METHOD PRIVATE popup : BOOL
VAR_INPUT
END_VAR
CASE popupStep OF
0:
	IF length>0 AND bSendCondition THEN
		_PopupLength:=length;
		popupSendData:=sendDataArray[cNumBegin];
		FOR iPopup:=cNumBegin TO (_PopupLength-1) DO
			sendDataArray[iPopup]:=sendDataArray[iPopup+1];
		END_FOR
		endPoint:=endPoint-1;
		length:=endPoint-cNumBegin;
		sendData(popupSendData);//此处是调用信息发送
		popupStep:=10;
	END_IF
10:
	popupTON2(IN:=NOT popupTON2.Q, PT:=T#2S);
	IF NOT bSendCondition OR popupTON2.Q THEN
		popupTON2(IN:=FALSE);
		popupStep:=11;
	END_IF
11:
	IF bSendCondition THEN
		popupStep:=12;
	END_IF
	popupTON1(IN:=FALSE);
12:
	//popupTON1(IN:=NOT popupTON1.Q,PT:=T#10MS);
	popupTON1(IN:=NOT popupTON1.Q,PT:=TO_TIME(nQueueInterval));
	IF popupTON1.Q THEN
		popupStep:=0;
	END_IF
END_CASE
END_METHOD

METHOD PRIVATE sendData : BOOL
VAR_INPUT
	dataStruct	:STRING(255);
END_VAR
IF bSendCondition AND bEnable THEN
	tcpipSendData:=dataStruct;
	
	CASE nSocketType OF
	0://TCPIP server
		tcpipSendDataBuff_Server:=tcpipSendData;
		tcpipSendData:=tcpipSendDataClear;	
		tcpipServer.bSend:=TRUE;
	1://TCPIP client
		tcpipSendDataBuff_Client:=tcpipSendData;
		tcpipSendData:=tcpipSendDataClear;	
		tcpipClient.bSend:=TRUE;
	END_CASE
	
	FOR logHandleArray_index:=1 TO logHandleArrayLength DO
		CASE nSocketType OF
		0://TCPIP server
			logHandleArray[logHandleArray_index]^.append(CONCAT(CONCAT(CONCAT('Send To ', sTerminalName), ' -- '),tcpipSendDataBuff_Server));
		1://TCPIP client
			logHandleArray[logHandleArray_index]^.append(CONCAT(CONCAT(CONCAT('Send To ', sTerminalName), ' -- '),tcpipSendDataBuff_Client));
		END_CASE
	END_FOR
END_IF
END_METHOD

END_PROGRAM

// ---- POUs/BaseModule/EL2252_2262Control/FlipperModule_EL2252.TcPOU
FUNCTION_BLOCK FlipperModule_EL2252
VAR CONSTANT
	gMaxPosNum								:INT:=100;
END_VAR
VAR_IN_OUT
	RefAxis_Ch1								:AXIS_REF;//ch1 运动主轴
	RemAxis_Ch1								:AXIS_REF;//ch1 锁存主轴
	RefAxis_Ch2								:AXIS_REF;//ch2 运动主轴
	RemAxis_Ch2								:AXIS_REF;//ch2 锁存主轴
END_VAR
VAR_INPUT
	FlipperOut1Times						:INT;//ch1 位置检测次数
	EnableOut1								:BOOL;//ch1 启用检测
	Out1_CamSwitchData						:ARRAY [1..gMaxPosNum] OF ST_CamSwitch;
	ForceOut1								:BOOL:=FALSE;//ch1 强制触发

	FlipperOut2Times						:INT;//ch2 位置检测次数
	EnableOut2								:BOOL;//ch2 启用检测
	ForceOut2								:BOOL:=FALSE;//ch2 强制触发
	Out2_CamSwitchData						:ARRAY [1..gMaxPosNum] OF ST_CamSwitch;
END_VAR
VAR_OUTPUT
	Out1RecPosArray1						:ARRAY [1..gMaxPosNum] OF LREAL:=[gMaxPosNum(0)];
	Out2RecPosArray2						:ARRAY [1..gMaxPosNum] OF LREAL:=[gMaxPosNum(0)];
	Ch1_LogOut								:STRING(255);
	Ch2_LogOut								:STRING(255);
	Io_EL2252								:EL2252_IoInterface;//硬件IO，需要关联至EL2252
	Ch1_Io_EL1252							:EL1252_IoInterface;//硬件IO，需要关联至EL1252
	Ch2_Io_EL1252							:EL1252_IoInterface;//硬件IO，需要关联至EL1252
END_VAR
VAR
//********************  XFC Calculate  *************************************************//
	Ch1_MC_DigitalCamSwitch					:MC_DigitalCamSwitch;
	Ch1_CAMSWITCH_REF						:CAMSWITCH_REF;
	Ch1_ArrMC_CamSwitch						:ARRAY [1..gMaxPosNum] OF MC_CamSwitch;
	Ch1_OUTPUT_REF							:OUTPUT_REF;
	Ch1_ST_CamSwitchOptions					:ST_CamSwitchOptions;
	Ch1_TRACK_REF							:TRACK_REF;

	Ch1_v									:INT:=0;//for CamswitchArray instance FirstPos and LastPos

	Ch2_MC_DigitalCamSwitch					:MC_DigitalCamSwitch;
	Ch2_CAMSWITCH_REF						:CAMSWITCH_REF;
	Ch2_ArrMC_CamSwitch						:ARRAY [1..gMaxPosNum] OF MC_CamSwitch;
	Ch2_OUTPUT_REF							:OUTPUT_REF;
	Ch2_ST_CamSwitchOptions					:ST_CamSwitchOptions;
	Ch2_TRACK_REF							:TRACK_REF;
	
	Ch2_v									:INT:=0;//for CamswitchArray instance FirstPos and LastPos
//********************  EL2252  *************************************************//
	Flipper_XFC_EL2252_V2					:XFC_EL2252_V2;
//****************************** XFC_touchprobe & EL1252  **********************//
	Ch1_XFC_TouchProbe						:XFC_TouchProbe;
	Ch1_ST_XfcTouchProbeOptions				:ST_XfcTouchProbeOptions;
	Ch1_XFC_TRIGGER_REF						:XFC_TRIGGER_REF;

	Ch1_fRecPos								:LREAL;
	Ch1_RecTrig								:R_TRIG;
	Ch1_nRecTimes							:INT:=1;
	Ch1_i									:INT:=1;

	Ch2_XFC_TouchProbe						:XFC_TouchProbe;
	Ch2_ST_XfcTouchProbeOptions				:ST_XfcTouchProbeOptions;
	Ch2_XFC_TRIGGER_REF						:XFC_TRIGGER_REF;

	Ch2_fRecPos								:LREAL;
	Ch2_RecTrig								:R_TRIG;
	Ch2_nRecTimes							:INT:=1;
	Ch2_i									:INT:=0;
	
	Ch1_LogFtrig							:F_TRIG;
	Ch1_LogRtrig							:R_TRIG;
	Ch1ClearI								:INT;
	Ch2_LogFtrig							:F_TRIG;
	Ch2_LogRtrig							:R_TRIG;
	Ch2ClearI								:INT;
END_VAR


//******************** Flipper Pos ****************************//
FOR Ch1_v:=1 TO FlipperOut1Times BY 1 DO
	Ch1_ArrMC_CamSwitch[Ch1_v].FirstOnPosition:=Out1_CamSwitchData[Ch1_v].fFirstOnPosition;
	Ch1_ArrMC_CamSwitch[Ch1_v].LastOnPosition:=Out1_CamSwitchData[Ch1_v].fLastOnPosition;//Out1PosS[Ch1_v]+1.5, Out1PosE[Ch1_v]
	
	IF Out1_CamSwitchData[Ch1_v].bTimeMode THEN
		Out1_CamSwitchData[Ch1_v].iAxisDirection:=0;
		Ch1_ArrMC_CamSwitch[Ch1_v].CamSwitchMode:=E_CamSwitchMode.CAMSWITCHMODE_TIME;//用时间模式可以通过 Duration 参数控制ON持续时间
		Ch1_ArrMC_CamSwitch[Ch1_v].Duration:=Out1_CamSwitchData[Ch1_v].fDuration;//持续时间, 单位s
	ELSE
		Ch1_ArrMC_CamSwitch[Ch1_v].CamSwitchMode:=E_CamSwitchMode.CAMSWITCHMODE_POSITION;//用位置模式可以通过 FirstOnPosition和LastOnPosition 参数控制ON持续时间
	END_IF
	IF 0>Out1_CamSwitchData[Ch1_v].iAxisDirection THEN
		Ch1_ArrMC_CamSwitch[Ch1_v].AxisDirection:=E_CamSwitchDirection.CAMSWITCHDIRECTION_NEGATIVE;
	ELSIF 0=Out1_CamSwitchData[Ch1_v].iAxisDirection THEN
		Ch1_ArrMC_CamSwitch[Ch1_v].AxisDirection:=E_CamSwitchDirection.CAMSWITCHDIRECTION_BOTH;
	ELSE
		Ch1_ArrMC_CamSwitch[Ch1_v].AxisDirection:=E_CamSwitchDirection.CAMSWITCHDIRECTION_POSITIVE;
	END_IF
END_FOR
Ch1_CAMSWITCH_REF.NumberOfSwitches:=TO_UDINT(FlipperOut1Times);
Ch1_CAMSWITCH_REF.pSwitches:=ADR(Ch1_ArrMC_CamSwitch);
Ch1_CAMSWITCH_REF.SizeOfSwitches:=SIZEOF(Ch1_ArrMC_CamSwitch);

FOR Ch2_v:=1 TO FlipperOut2Times BY 1 DO
	Ch2_ArrMC_CamSwitch[Ch2_v].FirstOnPosition:=Out2_CamSwitchData[Ch2_v].fFirstOnPosition;
	Ch2_ArrMC_CamSwitch[Ch2_v].LastOnPosition:=Out2_CamSwitchData[Ch2_v].fLastOnPosition;//Out2PosS[Ch2_v]+1.5, Out2PosE[Ch2_v]
	
	IF Out2_CamSwitchData[Ch2_v].bTimeMode THEN
		Out2_CamSwitchData[Ch2_v].iAxisDirection:=0;
		Ch2_ArrMC_CamSwitch[Ch2_v].CamSwitchMode:=E_CamSwitchMode.CAMSWITCHMODE_TIME;//用时间模式可以通过 Duration 参数控制ON持续时间
		Ch2_ArrMC_CamSwitch[Ch2_v].Duration:=Out2_CamSwitchData[Ch2_v].fDuration;//持续时间, 单位s
	ELSE
		Ch2_ArrMC_CamSwitch[Ch2_v].CamSwitchMode:=E_CamSwitchMode.CAMSWITCHMODE_POSITION;//用位置模式可以通过 FirstOnPosition和LastOnPosition 参数控制ON持续时间
	END_IF
	IF 0>Out2_CamSwitchData[Ch2_v].iAxisDirection THEN
		Ch2_ArrMC_CamSwitch[Ch2_v].AxisDirection:=E_CamSwitchDirection.CAMSWITCHDIRECTION_NEGATIVE;
	ELSIF 0=Out2_CamSwitchData[Ch2_v].iAxisDirection THEN
		Ch2_ArrMC_CamSwitch[Ch2_v].AxisDirection:=E_CamSwitchDirection.CAMSWITCHDIRECTION_BOTH;
	ELSE
		Ch2_ArrMC_CamSwitch[Ch2_v].AxisDirection:=E_CamSwitchDirection.CAMSWITCHDIRECTION_POSITIVE;
	END_IF
END_FOR
Ch2_CAMSWITCH_REF.NumberOfSwitches:=TO_UDINT(FlipperOut2Times);
Ch2_CAMSWITCH_REF.pSwitches:=ADR(Ch2_ArrMC_CamSwitch);
Ch2_CAMSWITCH_REF.SizeOfSwitches:=SIZEOF(Ch2_ArrMC_CamSwitch);
//******************** Cyclic IO ****************************//
EL1252();
EL2252V2();

METHOD PRIVATE EL1252
VAR_INPUT
END_VAR
//****************************** out1 EL1252 ***************************************//
Ch1_ST_XfcTouchProbeOptions.UseAcceleration:=TRUE;

Ch1_XFC_TRIGGER_REF.Signal:=Ch1_Io_EL1252.Input;
Ch1_XFC_TRIGGER_REF.TimestampRisingEdge:=Ch1_Io_EL1252.TimeStampNeg.dwLowPart;
Ch1_XFC_TRIGGER_REF.TimestampFallingEdge:=Ch1_Io_EL1252.TimeStampPos.dwLowPart;
Ch1_XFC_TRIGGER_REF.Edge:=E_SignalEdge.FallingEdge;
Ch1_XFC_TRIGGER_REF.FreeRun:=TRUE;
Ch1_XFC_TRIGGER_REF.ModuloPositions:=FALSE;
Ch1_XFC_TRIGGER_REF.EncoderIndex:=0;//DWORD_TO_UINT(RemAxis.NcToPlc.AxisId);

Ch1_XFC_TouchProbe(
	Axis:=RemAxis_Ch1 , 
	TriggerInput:=Ch1_XFC_TRIGGER_REF , 
	Execute:=TRUE , 
	WindowOnly:=FALSE , 
	FirstPosition:=0 , 
	LastPosition:=0 , 
	Options:=Ch1_ST_XfcTouchProbeOptions , 
	Done=> , 
	Busy=> , 
	Error=> , 
	ErrorID=> , 
	RecordedPosition=>Ch1_fRecPos );

Ch1_RecTrig(clk:=Ch1_XFC_TouchProbe.Done);
IF EnableOut1 THEN
	IF Ch1_RecTrig.Q THEN
		out1RecPosArray1[Ch1_nRecTimes]:=Ch1_fRecPos;
		Ch1_nRecTimes:=Ch1_nRecTimes+1;
	END_IF
END_IF

Ch1_LogRtrig(clk:=EnableOut1);
IF Ch1_LogRtrig.Q THEN
	FOR Ch1ClearI:=1 TO gMaxPosNum DO
		out1RecPosArray1[Ch1ClearI]:=0;
	END_FOR
END_IF

Ch1_LogFtrig(clk:=EnableOut1);
IF Ch1_LogFtrig.Q THEN
	Ch1_LogOut:='out1 Pos: ';
	FOR Ch1_i:=1 TO FlipperOut1Times BY 1 DO
		Ch1_LogOut:=concat(Ch1_LogOut,LREAL_TO_STRING(out1RecPosArray1[Ch1_i]));
		Ch1_LogOut:=concat(Ch1_LogOut,' ');
	END_FOR
	Ch1_nRecTimes:=1;
END_IF
//****************************** out2 EL1252 ***************************************//
Ch2_ST_XfcTouchProbeOptions.UseAcceleration:=TRUE;

Ch2_XFC_TRIGGER_REF.Signal:=Ch2_Io_EL1252.Input;
Ch2_XFC_TRIGGER_REF.TimestampRisingEdge:=Ch2_Io_EL1252.TimeStampNeg.dwLowPart;
Ch2_XFC_TRIGGER_REF.TimestampFallingEdge:=Ch2_Io_EL1252.TimeStampPos.dwLowPart;
Ch2_XFC_TRIGGER_REF.Edge:=E_SignalEdge.FallingEdge;
Ch2_XFC_TRIGGER_REF.FreeRun:=TRUE;
Ch2_XFC_TRIGGER_REF.ModuloPositions:=FALSE;
Ch2_XFC_TRIGGER_REF.EncoderIndex:=0;//DWORD_TO_UINT(RemAxis.NcToPlc.AxisId);

Ch2_XFC_TouchProbe(
	Axis:=RemAxis_Ch2 , 
	TriggerInput:=Ch2_XFC_TRIGGER_REF , 
	Execute:=TRUE , 
	WindowOnly:=FALSE , 
	FirstPosition:=0 , 
	LastPosition:=0 , 
	Options:=Ch2_ST_XfcTouchProbeOptions , 
	Done=> , 
	Busy=> , 
	Error=> , 
	ErrorID=> , 
	RecordedPosition=>Ch2_fRecPos );

Ch2_RecTrig(clk:=Ch2_XFC_TouchProbe.Done);
IF EnableOut2 THEN
	IF Ch2_RecTrig.Q THEN
		out2RecPosArray2[Ch2_nRecTimes]:=Ch2_fRecPos;
		Ch2_nRecTimes:=Ch2_nRecTimes+1;
	END_IF
END_IF

Ch2_LogRtrig(clk:=EnableOut2);
IF Ch2_LogRtrig.Q THEN
	FOR Ch2ClearI:=1 TO gMaxPosNum DO
		Out2RecPosArray2[Ch2ClearI]:=0;
	END_FOR
END_IF

Ch2_LogFtrig(clk:=EnableOut2);
IF Ch2_LogFtrig.Q THEN
	Ch2_LogOut:='out2 Pos: ';
	FOR Ch2_i:=1 TO FlipperOut2Times BY 1 DO
		Ch2_LogOut:=concat(Ch2_LogOut,LREAL_TO_STRING(out2RecPosArray2[Ch2_i]));
		Ch2_LogOut:=concat(Ch2_LogOut,' ');
	END_FOR
	Ch2_nRecTimes:=1;
END_IF
END_METHOD

METHOD PRIVATE EL2252V2
VAR_INPUT
END_VAR
//*******************   output 1  *****************************//
Ch1_ST_CamSwitchOptions.EncoderIndex:=0;//DWORD_TO_UINT(RefAxis.NcToPlc.AxisId);
Ch1_ST_CamSwitchOptions.UseAcceleration:=TRUE;

Ch1_TRACK_REF.ModuloPositions:=FALSE;//启用 模位置
Ch1_TRACK_REF.Disable:=FALSE;
Ch1_TRACK_REF.Force:=ForceOut1;
Ch1_TRACK_REF.OnCompensation:=0;//延时 ON
Ch1_TRACK_REF.OffCompensation:=0;//延时 OFF

Ch1_MC_DigitalCamSwitch(
	Axis:=RefAxis_Ch1 , 
	Switches:=Ch1_CAMSWITCH_REF , 
	Output:=Ch1_OUTPUT_REF , 
	TrackOptions:=Ch1_TRACK_REF , 
	Enable:=EnableOut1 , 
	Options:=Ch1_ST_CamSwitchOptions , 
	InOperation=> , 
	Busy=> , 
	Error=> , 
	ErrorID=> );

//*******************   output 2  *****************************//
Ch2_ST_CamSwitchOptions.EncoderIndex:=0;//DWORD_TO_UINT(RefAxis.NcToPlc.AxisId);
Ch2_ST_CamSwitchOptions.UseAcceleration:=TRUE;

Ch2_TRACK_REF.ModuloPositions:=FALSE;//启用 模位置
Ch2_TRACK_REF.Disable:=FALSE;
Ch2_TRACK_REF.Force:=ForceOut2;
Ch2_TRACK_REF.OnCompensation:=0;//延时 ON
Ch2_TRACK_REF.OffCompensation:=0;//延时 OFF

Ch2_MC_DigitalCamSwitch(
	Axis:=RefAxis_Ch2 , 
	Switches:=Ch2_CAMSWITCH_REF , 
	Output:=Ch2_OUTPUT_REF , 
	TrackOptions:=Ch2_TRACK_REF , 
	Enable:=EnableOut2 , 
	Options:=Ch2_ST_CamSwitchOptions , 
	InOperation=> , 
	Busy=> , 
	Error=> , 
	ErrorID=> );

//***************** EL2252 *****************************//
Flipper_XFC_EL2252_V2(
	ForceWhenLate:=TRUE , 
	Error=> , 
	ErrorID=> , 
	ErrorOutputMissed=> , 
	PrecisionReduced=> , 
	Output1:=Ch1_OUTPUT_REF , 
	Output2:=Ch2_OUTPUT_REF , 
	TrackOptions1:=Ch1_TRACK_REF , 
	TrackOptions2:=Ch2_TRACK_REF , 
	EL2252:=Io_EL2252 );
END_METHOD

METHOD SetCamSwitchData_Ch1 : BOOL
VAR_INPUT
	nIndex:INT;
	
	bTimeMode:BOOL;//TRUE表示时间控制模式, 持续时间由fDuration控制; FALSE表示位置控制模式，持续时间由fFirstOnPosition和fLastOnPosition控制
	fDuration:LREAL;//持续时间, 单位s
	
	fFirstOnPosition:LREAL;//时间控制模式和位置控制模式触发起始点
	fLastOnPosition:LREAL;//位置控制模式触发结束点
	iAxisDirection:INT;//-1表示负方向检测; 0表示正负方向检测(时间控制模式必须是0); 1表示正方向检测;
END_VAR
IF nIndex<1 OR nIndex>gMaxPosNum THEN
	SetCamSwitchData_Ch1:=FALSE;
	RETURN;
END_IF
Out1_CamSwitchData[nIndex].bTimeMode:=bTimeMode;
Out1_CamSwitchData[nIndex].fDuration:=fDuration;
Out1_CamSwitchData[nIndex].fFirstOnPosition:=fFirstOnPosition;
Out1_CamSwitchData[nIndex].fLastOnPosition:=fLastOnPosition;
Out1_CamSwitchData[nIndex].iAxisDirection:=iAxisDirection;
SetCamSwitchData_Ch1:=TRUE;
END_METHOD

METHOD SetCamSwitchData_Ch2 : BOOL
VAR_INPUT
	nIndex:INT;
	
	bTimeMode:BOOL;//TRUE表示时间控制模式, 持续时间由fDuration控制; FALSE表示位置控制模式，持续时间由fFirstOnPosition和fLastOnPosition控制
	fDuration:LREAL;//持续时间, 单位s
	
	fFirstOnPosition:LREAL;//时间控制模式和位置控制模式触发起始点
	fLastOnPosition:LREAL;//位置控制模式触发结束点
	iAxisDirection:INT;//-1表示负方向检测; 0表示正负方向检测(时间控制模式必须是0); 1表示正方向检测;
END_VAR
IF nIndex<1 OR nIndex>gMaxPosNum THEN
	SetCamSwitchData_Ch2:=FALSE;
	RETURN;
END_IF
Out2_CamSwitchData[nIndex].bTimeMode:=bTimeMode;
Out2_CamSwitchData[nIndex].fDuration:=fDuration;
Out2_CamSwitchData[nIndex].fFirstOnPosition:=fFirstOnPosition;
Out2_CamSwitchData[nIndex].fLastOnPosition:=fLastOnPosition;
Out2_CamSwitchData[nIndex].iAxisDirection:=iAxisDirection;
SetCamSwitchData_Ch2:=TRUE;
END_METHOD

ACTION VersionLog:
(*
版本: V1.0.0.0
说明:
	1. 首个版本
/**************************************************/
版本: V1.0.0.1
说明:
	1. 增加触发上升沿清空EL1252位置记录数据
/**************************************************/
版本: V1.0.0.2
说明:
	1. 增加函数接口，用于设置飞拍监控数据
/**************************************************/
*)
END_ACTION

END_FUNCTION_BLOCK

// ---- POUs/BaseModule/EL2252_2262Control/FlipperModule_EL2262.TcPOU
FUNCTION_BLOCK FlipperModule_EL2262
VAR CONSTANT
	gMaxPosNum								:INT:=100;
END_VAR
VAR_IN_OUT
	RefAxis_Ch1								:AXIS_REF;//ch1 运动主轴
	RemAxis_Ch1								:AXIS_REF;//ch1 锁存主轴
	RefAxis_Ch2								:AXIS_REF;//ch2 运动主轴
	RemAxis_Ch2								:AXIS_REF;//ch2 锁存主轴
END_VAR
VAR_INPUT
	OversamplingFactor						:UINT:=1000;// 超采样因子, Operation Mode需要设置成2 Channels(Bytes)
	FlipperOut1Times						:INT;//ch1 位置检测次数
	EnableOut1								:BOOL;//ch1 启用检测
	Out1_CamSwitchData						:ARRAY [1..gMaxPosNum] OF ST_CamSwitch_EL2262;
	ForceOut1								:BOOL:=FALSE;//ch1 强制触发

	FlipperOut2Times						:INT;//ch2 位置检测次数
	EnableOut2								:BOOL;//ch2 启用检测
	Out2_CamSwitchData						:ARRAY [1..gMaxPosNum] OF ST_CamSwitch_EL2262;
	ForceOut2								:BOOL:=FALSE;//ch2 强制触发
END_VAR
VAR_OUTPUT
	Out1RecPosArray1						:ARRAY [1..gMaxPosNum] OF LREAL:=[gMaxPosNum(0)];//记录锁存触发位置数组
	Out2RecPosArray2						:ARRAY [1..gMaxPosNum] OF LREAL:=[gMaxPosNum(0)];//记录锁存触发位置数组
	Ch1_LogOut								:STRING(255);
	Ch2_LogOut								:STRING(255);
	Io_EL2262								:EL2262_IoInterface;//硬件IO，需要关联至EL2262
	Io_EL2262_Ch2							:EL2262_IoInterface;//硬件IO，需要关联至EL2262
	Ch1_Io_EL1252							:EL1252_IoInterface;//硬件IO，需要关联至EL1252
	Ch2_Io_EL1252							:EL1252_IoInterface;//硬件IO，需要关联至EL1252
END_VAR
VAR
//********************  XFC Calculate  *************************************************//
	Ch1_MC_DigitalCamSwitch					:MC_DigitalCamSwitch;
	Ch1_CAMSWITCH_REF						:CAMSWITCH_REF;
	Ch1_ArrMC_CamSwitch						:ARRAY [1..gMaxPosNum] OF MC_CamSwitch;
	Ch1_OUTPUT_REF							:OUTPUT_REF;
	Ch1_ST_CamSwitchOptions					:ST_CamSwitchOptions;
	Ch1_TRACK_REF							:TRACK_REF;

	Ch1_v									:INT:=0;//for CamswitchArray instance FirstPos and LastPos

	Ch2_MC_DigitalCamSwitch					:MC_DigitalCamSwitch;
	Ch2_CAMSWITCH_REF						:CAMSWITCH_REF;
	Ch2_ArrMC_CamSwitch						:ARRAY [1..gMaxPosNum] OF MC_CamSwitch;
	Ch2_OUTPUT_REF							:OUTPUT_REF;
	Ch2_ST_CamSwitchOptions					:ST_CamSwitchOptions;
	Ch2_TRACK_REF							:TRACK_REF;
	
	Ch2_v									:INT:=0;//for CamswitchArray instance FirstPos and LastPos
//********************  EL2252  *************************************************//
	Flipper_CH1_XFC_EL2262					:XFC_EL2262;
	Flipper_CH2_XFC_EL2262					:XFC_EL2262;
	
//****************************** XFC_touchprobe & EL1252  **********************//
	Ch1_XFC_TouchProbe						:XFC_TouchProbe;
	Ch1_ST_XfcTouchProbeOptions				:ST_XfcTouchProbeOptions;
	Ch1_XFC_TRIGGER_REF						:XFC_TRIGGER_REF;

	Ch1_fRecPos								:LREAL;
	Ch1_RecTrig								:R_TRIG;
	Ch1_nRecTimes							:INT:=1;//用于记录锁存触发次数
	Ch1_i									:INT:=1;

	Ch2_XFC_TouchProbe						:XFC_TouchProbe;
	Ch2_ST_XfcTouchProbeOptions				:ST_XfcTouchProbeOptions;
	Ch2_XFC_TRIGGER_REF						:XFC_TRIGGER_REF;

	Ch2_fRecPos								:LREAL;
	Ch2_RecTrig								:R_TRIG;
	Ch2_nRecTimes							:INT:=1;//用于记录锁存触发次数
	Ch2_i									:INT:=0;
	
	Ch1_LogFtrig							:F_TRIG;
	Ch1_LogRtrig							:R_TRIG;
	Ch1ClearI								:INT;
	Ch2_LogFtrig							:F_TRIG;
	Ch2_LogRtrig							:R_TRIG;
	Ch2ClearI								:INT;
END_VAR


//******************** Flipper Pos ****************************//
FOR Ch1_v:=1 TO FlipperOut1Times BY 1 DO
	Ch1_ArrMC_CamSwitch[Ch1_v].FirstOnPosition:=Out1_CamSwitchData[Ch1_v].fFirstOnPosition;
	Ch1_ArrMC_CamSwitch[Ch1_v].LastOnPosition:=Out1_CamSwitchData[Ch1_v].fLastOnPosition;//Out1PosS[Ch1_v]+1.5, Out1PosE[Ch1_v]
	
	IF Out1_CamSwitchData[Ch1_v].bTimeMode THEN
		Out1_CamSwitchData[Ch1_v].iAxisDirection:=0;
		Ch1_ArrMC_CamSwitch[Ch1_v].CamSwitchMode:=E_CamSwitchMode.CAMSWITCHMODE_TIME;//用时间模式可以通过 Duration 参数控制ON持续时间
		Ch1_ArrMC_CamSwitch[Ch1_v].Duration:=Out1_CamSwitchData[Ch1_v].fDuration;//持续时间, 单位s
	ELSE
		Ch1_ArrMC_CamSwitch[Ch1_v].CamSwitchMode:=E_CamSwitchMode.CAMSWITCHMODE_POSITION;//用位置模式可以通过 FirstOnPosition和LastOnPosition 参数控制ON持续时间
	END_IF
	IF 0>Out1_CamSwitchData[Ch1_v].iAxisDirection THEN
		Ch1_ArrMC_CamSwitch[Ch1_v].AxisDirection:=E_CamSwitchDirection.CAMSWITCHDIRECTION_NEGATIVE;
	ELSIF 0=Out1_CamSwitchData[Ch1_v].iAxisDirection THEN
		Ch1_ArrMC_CamSwitch[Ch1_v].AxisDirection:=E_CamSwitchDirection.CAMSWITCHDIRECTION_BOTH;
	ELSE
		Ch1_ArrMC_CamSwitch[Ch1_v].AxisDirection:=E_CamSwitchDirection.CAMSWITCHDIRECTION_POSITIVE;
	END_IF
	
	(*Ch1_ArrMC_CamSwitch[Ch1_v].CamSwitchMode:=E_CamSwitchMode.CAMSWITCHMODE_POSITION;//用位置模式可以通过 FirstOnPosition和LastOnPosition 参数控制ON持续时间
	IF 0>Out1_CamSwitchData[Ch1_v].iAxisDirection THEN
		Ch1_ArrMC_CamSwitch[Ch1_v].AxisDirection:=E_CamSwitchDirection.CAMSWITCHDIRECTION_NEGATIVE;
	ELSIF 0=Out1_CamSwitchData[Ch1_v].iAxisDirection THEN
		Ch1_ArrMC_CamSwitch[Ch1_v].AxisDirection:=E_CamSwitchDirection.CAMSWITCHDIRECTION_BOTH;
	ELSE
		Ch1_ArrMC_CamSwitch[Ch1_v].AxisDirection:=E_CamSwitchDirection.CAMSWITCHDIRECTION_POSITIVE;
	END_IF*)
END_FOR
Ch1_CAMSWITCH_REF.NumberOfSwitches:=TO_UDINT(FlipperOut1Times);
Ch1_CAMSWITCH_REF.pSwitches:=ADR(Ch1_ArrMC_CamSwitch);
Ch1_CAMSWITCH_REF.SizeOfSwitches:=SIZEOF(Ch1_ArrMC_CamSwitch);

FOR Ch2_v:=1 TO FlipperOut2Times BY 1 DO
	Ch2_ArrMC_CamSwitch[Ch2_v].FirstOnPosition:=Out2_CamSwitchData[Ch2_v].fFirstOnPosition;
	Ch2_ArrMC_CamSwitch[Ch2_v].LastOnPosition:=Out2_CamSwitchData[Ch2_v].fLastOnPosition;//Out2PosS[Ch2_v]+1.5, Out2PosE[Ch2_v]
	
	IF Out2_CamSwitchData[Ch2_v].bTimeMode THEN
		Out2_CamSwitchData[Ch2_v].iAxisDirection:=0;
		Ch2_ArrMC_CamSwitch[Ch2_v].CamSwitchMode:=E_CamSwitchMode.CAMSWITCHMODE_TIME;//用时间模式可以通过 Duration 参数控制ON持续时间
		Ch2_ArrMC_CamSwitch[Ch2_v].Duration:=Out2_CamSwitchData[Ch2_v].fDuration;//持续时间, 单位s
	ELSE
		Ch2_ArrMC_CamSwitch[Ch2_v].CamSwitchMode:=E_CamSwitchMode.CAMSWITCHMODE_POSITION;//用位置模式可以通过 FirstOnPosition和LastOnPosition 参数控制ON持续时间
	END_IF
	IF 0>Out2_CamSwitchData[Ch2_v].iAxisDirection THEN
		Ch2_ArrMC_CamSwitch[Ch2_v].AxisDirection:=E_CamSwitchDirection.CAMSWITCHDIRECTION_NEGATIVE;
	ELSIF 0=Out2_CamSwitchData[Ch2_v].iAxisDirection THEN
		Ch2_ArrMC_CamSwitch[Ch2_v].AxisDirection:=E_CamSwitchDirection.CAMSWITCHDIRECTION_BOTH;
	ELSE
		Ch2_ArrMC_CamSwitch[Ch2_v].AxisDirection:=E_CamSwitchDirection.CAMSWITCHDIRECTION_POSITIVE;
	END_IF
	
	(*Ch2_ArrMC_CamSwitch[Ch2_v].CamSwitchMode:=E_CamSwitchMode.CAMSWITCHMODE_POSITION;//用位置模式可以通过 FirstOnPosition和LastOnPosition 参数控制ON持续时间
	IF 0>Out2_CamSwitchData[Ch2_v].iAxisDirection THEN
		Ch2_ArrMC_CamSwitch[Ch2_v].AxisDirection:=E_CamSwitchDirection.CAMSWITCHDIRECTION_NEGATIVE;
	ELSIF 0=Out2_CamSwitchData[Ch2_v].iAxisDirection THEN
		Ch2_ArrMC_CamSwitch[Ch2_v].AxisDirection:=E_CamSwitchDirection.CAMSWITCHDIRECTION_BOTH;
	ELSE
		Ch2_ArrMC_CamSwitch[Ch2_v].AxisDirection:=E_CamSwitchDirection.CAMSWITCHDIRECTION_POSITIVE;
	END_IF*)
END_FOR
Ch2_CAMSWITCH_REF.NumberOfSwitches:=TO_UDINT(FlipperOut2Times);
Ch2_CAMSWITCH_REF.pSwitches:=ADR(Ch2_ArrMC_CamSwitch);
Ch2_CAMSWITCH_REF.SizeOfSwitches:=SIZEOF(Ch2_ArrMC_CamSwitch);
//******************** Cyclic IO ****************************//
EL2262();
EL1252();

METHOD PRIVATE EL1252
VAR_INPUT
END_VAR
//****************************** out1 EL1252 ***************************************//
Ch1_ST_XfcTouchProbeOptions.UseAcceleration:=TRUE;
(*
Ch1_XFC_TRIGGER_REF.Signal:=Ch1_Io_EL1252.Input;
Ch1_XFC_TRIGGER_REF.TimestampRisingEdge:=Ch1_Io_EL1252.TimeStampNeg.dwLowPart;
Ch1_XFC_TRIGGER_REF.TimestampFallingEdge:=Ch1_Io_EL1252.TimeStampPos.dwLowPart;
Ch1_XFC_TRIGGER_REF.Edge:=E_SignalEdge.FallingEdge;
Ch1_XFC_TRIGGER_REF.FreeRun:=TRUE;
Ch1_XFC_TRIGGER_REF.ModuloPositions:=FALSE;
Ch1_XFC_TRIGGER_REF.EncoderIndex:=0;//DWORD_TO_UINT(RemAxis.NcToPlc.AxisId);
*)
Ch1_XFC_TRIGGER_REF.Signal:=Ch1_Io_EL1252.Input;
Ch1_XFC_TRIGGER_REF.TimestampRisingEdge:=Ch1_Io_EL1252.TimeStampPos.dwLowPart;
Ch1_XFC_TRIGGER_REF.TimestampFallingEdge:=Ch1_Io_EL1252.TimeStampNeg.dwLowPart;
Ch1_XFC_TRIGGER_REF.Edge:=E_SignalEdge.RisingEdge;
Ch1_XFC_TRIGGER_REF.FreeRun:=TRUE;
Ch1_XFC_TRIGGER_REF.ModuloPositions:=FALSE;
Ch1_XFC_TRIGGER_REF.EncoderIndex:=0;//DWORD_TO_UINT(RemAxis_Ch1.NcToPlc.AxisId);

RemAxis_Ch1.ReadStatus();
Ch1_XFC_TouchProbe(
	Axis:=RemAxis_Ch1 , 
	TriggerInput:=Ch1_XFC_TRIGGER_REF , 
	Execute:=TRUE , 
	WindowOnly:=FALSE , 
	FirstPosition:=0 , 
	LastPosition:=0 , 
	Options:=Ch1_ST_XfcTouchProbeOptions , 
	Done=> , 
	Busy=> , 
	Error=> , 
	ErrorID=> , 
	RecordedPosition=>Ch1_fRecPos );

Ch1_RecTrig(clk:=Ch1_XFC_TouchProbe.Done);
IF EnableOut1 THEN
	IF Ch1_RecTrig.Q THEN
		out1RecPosArray1[Ch1_nRecTimes]:=Ch1_fRecPos;
		Ch1_nRecTimes:=Ch1_nRecTimes+1;
	END_IF
END_IF

Ch1_LogRtrig(clk:=EnableOut1);
IF Ch1_LogRtrig.Q THEN
	FOR Ch1ClearI:=1 TO gMaxPosNum DO
		out1RecPosArray1[Ch1ClearI]:=0;
	END_FOR
END_IF

Ch1_LogFtrig(clk:=EnableOut1);
IF Ch1_LogFtrig.Q THEN
	Ch1_LogOut:='out1 Pos:,';
	//FOR Ch1_i:=1 TO FlipperOut1Times BY 1 DO
	FOR Ch1_i:=1 TO (Ch1_nRecTimes-1) BY 1 DO
		//Ch1_LogOut:=concat(Ch1_LogOut,LREAL_TO_STRING(out1RecPosArray1[Ch1_i]));
		Ch1_LogOut:=concat(Ch1_LogOut,LREAL_TO_FMTSTR(out1RecPosArray1[Ch1_i],5,FALSE));
		Ch1_LogOut:=concat(Ch1_LogOut,',');
	END_FOR
	Ch1_nRecTimes:=1;
END_IF
//****************************** out2 EL1252 ***************************************//
Ch2_ST_XfcTouchProbeOptions.UseAcceleration:=TRUE;
(*
Ch2_XFC_TRIGGER_REF.Signal:=Ch2_Io_EL1252.Input;
Ch2_XFC_TRIGGER_REF.TimestampRisingEdge:=Ch2_Io_EL1252.TimeStampNeg.dwLowPart;
Ch2_XFC_TRIGGER_REF.TimestampFallingEdge:=Ch2_Io_EL1252.TimeStampPos.dwLowPart;
Ch2_XFC_TRIGGER_REF.Edge:=E_SignalEdge.FallingEdge;
Ch2_XFC_TRIGGER_REF.FreeRun:=TRUE;
Ch2_XFC_TRIGGER_REF.ModuloPositions:=FALSE;
Ch2_XFC_TRIGGER_REF.EncoderIndex:=0;//DWORD_TO_UINT(RemAxis.NcToPlc.AxisId);
*)
Ch2_XFC_TRIGGER_REF.Signal:=Ch2_Io_EL1252.Input;
Ch2_XFC_TRIGGER_REF.TimestampRisingEdge:=Ch2_Io_EL1252.TimeStampPos.dwLowPart;
Ch2_XFC_TRIGGER_REF.TimestampFallingEdge:=Ch2_Io_EL1252.TimeStampNeg.dwLowPart;
Ch2_XFC_TRIGGER_REF.Edge:=E_SignalEdge.RisingEdge;
Ch2_XFC_TRIGGER_REF.FreeRun:=TRUE;
Ch2_XFC_TRIGGER_REF.ModuloPositions:=FALSE;
Ch2_XFC_TRIGGER_REF.EncoderIndex:=0;//DWORD_TO_UINT(RemAxis_Ch2.NcToPlc.AxisId);

RemAxis_Ch2.ReadStatus();
Ch2_XFC_TouchProbe(
	Axis:=RemAxis_Ch2 , 
	TriggerInput:=Ch2_XFC_TRIGGER_REF , 
	Execute:=TRUE , 
	WindowOnly:=FALSE , 
	FirstPosition:=0 , 
	LastPosition:=0 , 
	Options:=Ch2_ST_XfcTouchProbeOptions , 
	Done=> , 
	Busy=> , 
	Error=> , 
	ErrorID=> , 
	RecordedPosition=>Ch2_fRecPos );


Ch2_RecTrig(clk:=Ch2_XFC_TouchProbe.Done);
IF EnableOut2 THEN
	IF Ch2_RecTrig.Q THEN
		out2RecPosArray2[Ch2_nRecTimes]:=Ch2_fRecPos;
		Ch2_nRecTimes:=Ch2_nRecTimes+1;
	END_IF
END_IF

Ch2_LogRtrig(clk:=EnableOut2);
IF Ch2_LogRtrig.Q THEN
	FOR Ch2ClearI:=1 TO gMaxPosNum DO
		Out2RecPosArray2[Ch2ClearI]:=0;
	END_FOR
END_IF

Ch2_LogFtrig(clk:=EnableOut2);
IF Ch2_LogFtrig.Q THEN
	Ch2_LogOut:='out2 Pos:,';
	//FOR Ch2_i:=1 TO FlipperOut2Times BY 1 DO
	FOR Ch2_i:=1 TO (Ch2_nRecTimes-1) BY 1 DO
		//Ch2_LogOut:=concat(Ch2_LogOut,LREAL_TO_STRING(out2RecPosArray2[Ch2_i]));
		Ch2_LogOut:=concat(Ch2_LogOut,LREAL_TO_FMTSTR(out2RecPosArray2[Ch2_i],5,FALSE));
		Ch2_LogOut:=concat(Ch2_LogOut,',');
	END_FOR
	Ch2_nRecTimes:=1;
END_IF
END_METHOD

METHOD PRIVATE EL2262
VAR_INPUT
END_VAR
//*******************   output 1  *****************************//
Ch1_ST_CamSwitchOptions.EncoderIndex:=0;//DWORD_TO_UINT(RefAxis.NcToPlc.AxisId);
Ch1_ST_CamSwitchOptions.UseAcceleration:=TRUE;//FALSE TRUE

Ch1_TRACK_REF.ModuloPositions:=FALSE;//启用 模位置
Ch1_TRACK_REF.Disable:=FALSE;
Ch1_TRACK_REF.Force:=ForceOut1;
Ch1_TRACK_REF.OnCompensation:=0;//延时 ON
Ch1_TRACK_REF.OffCompensation:=0;//延时 OFF

RefAxis_Ch1.ReadStatus();
Ch1_MC_DigitalCamSwitch(
	Axis:=RefAxis_Ch1 , 
	Switches:=Ch1_CAMSWITCH_REF , 
	Output:=Ch1_OUTPUT_REF , 
	TrackOptions:=Ch1_TRACK_REF , 
	Enable:=EnableOut1 , 
	Options:=Ch1_ST_CamSwitchOptions , 
	InOperation=> , 
	Busy=> , 
	Error=> , 
	ErrorID=> );
(*
IF RefAxis_Ch1.Status.NotMoving THEN
	Ch1_MC_DigitalCamSwitch(
		Axis:=RefAxis_Ch1 , 
		Switches:=Ch1_CAMSWITCH_REF , 
		Output:=Ch1_OUTPUT_REF , 
		TrackOptions:=Ch1_TRACK_REF , 
		Enable:=FALSE , 
		Options:=Ch1_ST_CamSwitchOptions , 
		InOperation=> , 
		Busy=> , 
		Error=> , 
		ErrorID=> );
END_IF
*)
//*******************   output 2  *****************************//
Ch2_ST_CamSwitchOptions.EncoderIndex:=0;//DWORD_TO_UINT(RefAxis.NcToPlc.AxisId);
Ch2_ST_CamSwitchOptions.UseAcceleration:=TRUE;//FALSE TRUE

Ch2_TRACK_REF.ModuloPositions:=FALSE;//启用 模位置
Ch2_TRACK_REF.Disable:=FALSE;
Ch2_TRACK_REF.Force:=ForceOut2;
Ch2_TRACK_REF.OnCompensation:=0;//延时 ON
Ch2_TRACK_REF.OffCompensation:=0;//延时 OFF

RefAxis_Ch2.ReadStatus();
Ch2_MC_DigitalCamSwitch(
	Axis:=RefAxis_Ch2 , 
	Switches:=Ch2_CAMSWITCH_REF , 
	Output:=Ch2_OUTPUT_REF , 
	TrackOptions:=Ch2_TRACK_REF , 
	Enable:=EnableOut2 , 
	Options:=Ch2_ST_CamSwitchOptions , 
	InOperation=> , 
	Busy=> , 
	Error=> , 
	ErrorID=> );
(*
IF RefAxis_Ch2.Status.NotMoving THEN
	Ch2_MC_DigitalCamSwitch(
		Axis:=RefAxis_Ch2 , 
		Switches:=Ch2_CAMSWITCH_REF , 
		Output:=Ch2_OUTPUT_REF , 
		TrackOptions:=Ch2_TRACK_REF , 
		Enable:=FALSE , 
		Options:=Ch2_ST_CamSwitchOptions , 
		InOperation=> , 
		Busy=> , 
		Error=> , 
		ErrorID=> );
END_IF
*)
//***************** EL2262 *****************************//
Flipper_CH1_XFC_EL2262(
	OversamplingFactor:= OversamplingFactor, 
	OutputOneCycleDelayed:= FALSE, 
	ForceWhenLate:= TRUE, 
	Channel:= 0, 
	Error=> , 
	ErrorID=> , 
	ErrorOutputMissed=> , 
	PrecisionReduced=> , 
	Output:= Ch1_OUTPUT_REF, 
	TrackOptions:= Ch1_TRACK_REF, 
	EL2262:= Io_EL2262);

Flipper_CH2_XFC_EL2262(
	OversamplingFactor:= OversamplingFactor, 
	OutputOneCycleDelayed:= FALSE, 
	ForceWhenLate:= TRUE, 
	Channel:= 1, 
	Error=> , 
	ErrorID=> , 
	ErrorOutputMissed=> , 
	PrecisionReduced=> , 
	Output:= Ch2_OUTPUT_REF, 
	TrackOptions:= Ch2_TRACK_REF, 
	EL2262:= Io_EL2262_Ch2);
END_METHOD

METHOD SetCamSwitchData_Ch1 : BOOL
VAR_INPUT
	nIndex:INT;
	
	bTimeMode:BOOL;//TRUE表示时间控制模式, 持续时间由fDuration控制; FALSE表示位置控制模式，持续时间由fFirstOnPosition和fLastOnPosition控制
	fDuration:LREAL;//持续时间, 单位s
	
	fFirstOnPosition:LREAL;//时间控制模式和位置控制模式触发起始点
	fLastOnPosition:LREAL;//位置控制模式触发结束点
	iAxisDirection:INT;//-1表示负方向检测; 0表示正负方向检测(时间控制模式必须是0); 1表示正方向检测;
END_VAR
IF nIndex<1 OR nIndex>gMaxPosNum THEN
	SetCamSwitchData_Ch1:=FALSE;
	RETURN;
END_IF
Out1_CamSwitchData[nIndex].bTimeMode:=bTimeMode;
Out1_CamSwitchData[nIndex].fDuration:=fDuration;
Out1_CamSwitchData[nIndex].fFirstOnPosition:=fFirstOnPosition;
Out1_CamSwitchData[nIndex].fLastOnPosition:=fLastOnPosition;
Out1_CamSwitchData[nIndex].iAxisDirection:=iAxisDirection;
SetCamSwitchData_Ch1:=TRUE;
END_METHOD

METHOD SetCamSwitchData_Ch2 : BOOL
VAR_INPUT
	nIndex:INT;
	
	bTimeMode:BOOL;//TRUE表示时间控制模式, 持续时间由fDuration控制; FALSE表示位置控制模式，持续时间由fFirstOnPosition和fLastOnPosition控制
	fDuration:LREAL;//持续时间, 单位s
	
	fFirstOnPosition:LREAL;//时间控制模式和位置控制模式触发起始点
	fLastOnPosition:LREAL;//位置控制模式触发结束点
	iAxisDirection:INT;//-1表示负方向检测; 0表示正负方向检测(时间控制模式必须是0); 1表示正方向检测;
END_VAR
IF nIndex<1 OR nIndex>gMaxPosNum THEN
	SetCamSwitchData_Ch2:=FALSE;
	RETURN;
END_IF
Out2_CamSwitchData[nIndex].bTimeMode:=bTimeMode;
Out2_CamSwitchData[nIndex].fDuration:=fDuration;
Out2_CamSwitchData[nIndex].fFirstOnPosition:=fFirstOnPosition;
Out2_CamSwitchData[nIndex].fLastOnPosition:=fLastOnPosition;
Out2_CamSwitchData[nIndex].iAxisDirection:=iAxisDirection;
SetCamSwitchData_Ch2:=TRUE;
END_METHOD

ACTION VersionLog:
(*
版本: V1.0.0.0
说明:
	1. 首个版本
/**************************************************/
版本: V1.0.0.1
说明:
	1. 增加触发上升沿清空EL1252位置记录数据
/**************************************************/
版本: V1.0.0.2
说明:
	1. 增加函数接口，用于设置飞拍监控数据
/**************************************************/
*)
END_ACTION

END_FUNCTION_BLOCK

// ---- POUs/BaseModule/EL2252_2262Control/FlipperModule_EL2262_old.TcPOU
FUNCTION_BLOCK FlipperModule_EL2262_old
VAR CONSTANT
	gMaxPosNum								:INT:=100;
END_VAR
VAR_IN_OUT
	RefAxis_Ch1								:AXIS_REF;//ch1 运动主轴
	RemAxis_Ch1								:AXIS_REF;//ch1 锁存主轴
	RefAxis_Ch2								:AXIS_REF;//ch2 运动主轴
	RemAxis_Ch2								:AXIS_REF;//ch2 锁存主轴
END_VAR
VAR_INPUT
	OversamplingFactor						:UINT:=1000;// 超采样因子, Operation Mode需要设置成2 Channels(Bytes)
	FlipperOut1Times						:INT;//ch1 位置检测次数
	EnableOut1								:BOOL;//ch1 启用检测
	Out1_CamSwitchData						:ARRAY [1..gMaxPosNum] OF ST_CamSwitch_EL2262;
	ForceOut1								:BOOL:=FALSE;//ch1 强制触发

	FlipperOut2Times						:INT;//ch2 位置检测次数
	EnableOut2								:BOOL;//ch2 启用检测
	Out2_CamSwitchData						:ARRAY [1..gMaxPosNum] OF ST_CamSwitch_EL2262;
	ForceOut2								:BOOL:=FALSE;//ch2 强制触发
END_VAR
VAR_OUTPUT
	Out1RecPosArray1						:ARRAY [1..gMaxPosNum] OF LREAL:=[gMaxPosNum(0)];//记录锁存触发位置数组
	Out2RecPosArray2						:ARRAY [1..gMaxPosNum] OF LREAL:=[gMaxPosNum(0)];//记录锁存触发位置数组
	Ch1_LogOut								:STRING(255);
	Ch2_LogOut								:STRING(255);
	Io_EL2262								:EL2262_IoInterface;//硬件IO，需要关联至EL2262
	Io_EL2262_Ch2							:EL2262_IoInterface;//硬件IO，需要关联至EL2262
	Ch1_Io_EL1252							:EL1252_IoInterface;//硬件IO，需要关联至EL1252
	Ch2_Io_EL1252							:EL1252_IoInterface;//硬件IO，需要关联至EL1252
END_VAR
VAR
//********************  XFC Calculate  *************************************************//
	Ch1_MC_DigitalCamSwitch					:MC_DigitalCamSwitch;
	Ch1_CAMSWITCH_REF						:CAMSWITCH_REF;
	Ch1_ArrMC_CamSwitch						:ARRAY [1..gMaxPosNum] OF MC_CamSwitch;
	Ch1_OUTPUT_REF							:OUTPUT_REF;
	Ch1_ST_CamSwitchOptions					:ST_CamSwitchOptions;
	Ch1_TRACK_REF							:TRACK_REF;

	Ch1_v									:INT:=0;//for CamswitchArray instance FirstPos and LastPos

	Ch2_MC_DigitalCamSwitch					:MC_DigitalCamSwitch;
	Ch2_CAMSWITCH_REF						:CAMSWITCH_REF;
	Ch2_ArrMC_CamSwitch						:ARRAY [1..gMaxPosNum] OF MC_CamSwitch;
	Ch2_OUTPUT_REF							:OUTPUT_REF;
	Ch2_ST_CamSwitchOptions					:ST_CamSwitchOptions;
	Ch2_TRACK_REF							:TRACK_REF;
	
	Ch2_v									:INT:=0;//for CamswitchArray instance FirstPos and LastPos
//********************  EL2252  *************************************************//
	Flipper_CH1_XFC_EL2262					:XFC_EL2262;
	Flipper_CH2_XFC_EL2262					:XFC_EL2262;
	
//****************************** XFC_touchprobe & EL1252  **********************//
	Ch1_XFC_TouchProbe						:XFC_TouchProbe;
	Ch1_ST_XfcTouchProbeOptions				:ST_XfcTouchProbeOptions;
	Ch1_XFC_TRIGGER_REF						:XFC_TRIGGER_REF;

	Ch1_fRecPos								:LREAL;
	Ch1_RecTrig								:R_TRIG;
	Ch1_nRecTimes							:INT:=1;//用于记录锁存触发次数
	Ch1_i									:INT:=1;

	Ch2_XFC_TouchProbe						:XFC_TouchProbe;
	Ch2_ST_XfcTouchProbeOptions				:ST_XfcTouchProbeOptions;
	Ch2_XFC_TRIGGER_REF						:XFC_TRIGGER_REF;

	Ch2_fRecPos								:LREAL;
	Ch2_RecTrig								:R_TRIG;
	Ch2_nRecTimes							:INT:=1;//用于记录锁存触发次数
	Ch2_i									:INT:=0;
	
	Ch1_LogFtrig							:F_TRIG;
	Ch1_LogRtrig							:R_TRIG;
	Ch1ClearI								:INT;
	Ch2_LogFtrig							:F_TRIG;
	Ch2_LogRtrig							:R_TRIG;
	Ch2ClearI								:INT;
END_VAR


//******************** Flipper Pos ****************************//
FOR Ch1_v:=1 TO FlipperOut1Times BY 1 DO
	Ch1_ArrMC_CamSwitch[Ch1_v].FirstOnPosition:=Out1_CamSwitchData[Ch1_v].fFirstOnPosition;
	Ch1_ArrMC_CamSwitch[Ch1_v].LastOnPosition:=Out1_CamSwitchData[Ch1_v].fLastOnPosition;//Out1PosS[Ch1_v]+1.5, Out1PosE[Ch1_v]
	
	Ch1_ArrMC_CamSwitch[Ch1_v].CamSwitchMode:=E_CamSwitchMode.CAMSWITCHMODE_POSITION;//用位置模式可以通过 FirstOnPosition和LastOnPosition 参数控制ON持续时间
	IF 0>Out1_CamSwitchData[Ch1_v].iAxisDirection THEN
		Ch1_ArrMC_CamSwitch[Ch1_v].AxisDirection:=E_CamSwitchDirection.CAMSWITCHDIRECTION_NEGATIVE;
	ELSIF 0=Out1_CamSwitchData[Ch1_v].iAxisDirection THEN
		Ch1_ArrMC_CamSwitch[Ch1_v].AxisDirection:=E_CamSwitchDirection.CAMSWITCHDIRECTION_BOTH;
	ELSE
		Ch1_ArrMC_CamSwitch[Ch1_v].AxisDirection:=E_CamSwitchDirection.CAMSWITCHDIRECTION_POSITIVE;
	END_IF
END_FOR
Ch1_CAMSWITCH_REF.NumberOfSwitches:=TO_UDINT(FlipperOut1Times);
Ch1_CAMSWITCH_REF.pSwitches:=ADR(Ch1_ArrMC_CamSwitch);
Ch1_CAMSWITCH_REF.SizeOfSwitches:=SIZEOF(Ch1_ArrMC_CamSwitch);

FOR Ch2_v:=1 TO FlipperOut2Times BY 1 DO
	Ch2_ArrMC_CamSwitch[Ch2_v].FirstOnPosition:=Out2_CamSwitchData[Ch2_v].fFirstOnPosition;
	Ch2_ArrMC_CamSwitch[Ch2_v].LastOnPosition:=Out2_CamSwitchData[Ch2_v].fLastOnPosition;//Out2PosS[Ch2_v]+1.5, Out2PosE[Ch2_v]
	
	Ch2_ArrMC_CamSwitch[Ch2_v].CamSwitchMode:=E_CamSwitchMode.CAMSWITCHMODE_POSITION;//用位置模式可以通过 FirstOnPosition和LastOnPosition 参数控制ON持续时间
	IF 0>Out2_CamSwitchData[Ch2_v].iAxisDirection THEN
		Ch2_ArrMC_CamSwitch[Ch2_v].AxisDirection:=E_CamSwitchDirection.CAMSWITCHDIRECTION_NEGATIVE;
	ELSIF 0=Out2_CamSwitchData[Ch2_v].iAxisDirection THEN
		Ch2_ArrMC_CamSwitch[Ch2_v].AxisDirection:=E_CamSwitchDirection.CAMSWITCHDIRECTION_BOTH;
	ELSE
		Ch2_ArrMC_CamSwitch[Ch2_v].AxisDirection:=E_CamSwitchDirection.CAMSWITCHDIRECTION_POSITIVE;
	END_IF
END_FOR
Ch2_CAMSWITCH_REF.NumberOfSwitches:=TO_UDINT(FlipperOut2Times);
Ch2_CAMSWITCH_REF.pSwitches:=ADR(Ch2_ArrMC_CamSwitch);
Ch2_CAMSWITCH_REF.SizeOfSwitches:=SIZEOF(Ch2_ArrMC_CamSwitch);
//******************** Cyclic IO ****************************//
EL2262();
EL1252();

METHOD PRIVATE EL1252
VAR_INPUT
END_VAR
//****************************** out1 EL1252 ***************************************//
Ch1_ST_XfcTouchProbeOptions.UseAcceleration:=TRUE;
(*
Ch1_XFC_TRIGGER_REF.Signal:=Ch1_Io_EL1252.Input;
Ch1_XFC_TRIGGER_REF.TimestampRisingEdge:=Ch1_Io_EL1252.TimeStampNeg.dwLowPart;
Ch1_XFC_TRIGGER_REF.TimestampFallingEdge:=Ch1_Io_EL1252.TimeStampPos.dwLowPart;
Ch1_XFC_TRIGGER_REF.Edge:=E_SignalEdge.FallingEdge;
Ch1_XFC_TRIGGER_REF.FreeRun:=TRUE;
Ch1_XFC_TRIGGER_REF.ModuloPositions:=FALSE;
Ch1_XFC_TRIGGER_REF.EncoderIndex:=0;//DWORD_TO_UINT(RemAxis.NcToPlc.AxisId);
*)
Ch1_XFC_TRIGGER_REF.Signal:=Ch1_Io_EL1252.Input;
Ch1_XFC_TRIGGER_REF.TimestampRisingEdge:=Ch1_Io_EL1252.TimeStampPos.dwLowPart;
Ch1_XFC_TRIGGER_REF.TimestampFallingEdge:=Ch1_Io_EL1252.TimeStampNeg.dwLowPart;
Ch1_XFC_TRIGGER_REF.Edge:=E_SignalEdge.RisingEdge;
Ch1_XFC_TRIGGER_REF.FreeRun:=TRUE;
Ch1_XFC_TRIGGER_REF.ModuloPositions:=FALSE;
Ch1_XFC_TRIGGER_REF.EncoderIndex:=0;//DWORD_TO_UINT(RemAxis_Ch1.NcToPlc.AxisId);

RemAxis_Ch1.ReadStatus();
Ch1_XFC_TouchProbe(
	Axis:=RemAxis_Ch1 , 
	TriggerInput:=Ch1_XFC_TRIGGER_REF , 
	Execute:=TRUE , 
	WindowOnly:=FALSE , 
	FirstPosition:=0 , 
	LastPosition:=0 , 
	Options:=Ch1_ST_XfcTouchProbeOptions , 
	Done=> , 
	Busy=> , 
	Error=> , 
	ErrorID=> , 
	RecordedPosition=>Ch1_fRecPos );

Ch1_RecTrig(clk:=Ch1_XFC_TouchProbe.Done);
IF EnableOut1 THEN
	IF Ch1_RecTrig.Q THEN
		out1RecPosArray1[Ch1_nRecTimes]:=Ch1_fRecPos;
		Ch1_nRecTimes:=Ch1_nRecTimes+1;
	END_IF
END_IF

Ch1_LogRtrig(clk:=EnableOut1);
IF Ch1_LogRtrig.Q THEN
	FOR Ch1ClearI:=1 TO gMaxPosNum DO
		out1RecPosArray1[Ch1ClearI]:=0;
	END_FOR
END_IF

Ch1_LogFtrig(clk:=EnableOut1);
IF Ch1_LogFtrig.Q THEN
	Ch1_LogOut:='out1 Pos:,';
	//FOR Ch1_i:=1 TO FlipperOut1Times BY 1 DO
	FOR Ch1_i:=1 TO (Ch1_nRecTimes-1) BY 1 DO
		//Ch1_LogOut:=concat(Ch1_LogOut,LREAL_TO_STRING(out1RecPosArray1[Ch1_i]));
		Ch1_LogOut:=concat(Ch1_LogOut,LREAL_TO_FMTSTR(out1RecPosArray1[Ch1_i],5,FALSE));
		Ch1_LogOut:=concat(Ch1_LogOut,',');
	END_FOR
	Ch1_nRecTimes:=1;
END_IF
//****************************** out2 EL1252 ***************************************//
Ch2_ST_XfcTouchProbeOptions.UseAcceleration:=TRUE;
(*
Ch2_XFC_TRIGGER_REF.Signal:=Ch2_Io_EL1252.Input;
Ch2_XFC_TRIGGER_REF.TimestampRisingEdge:=Ch2_Io_EL1252.TimeStampNeg.dwLowPart;
Ch2_XFC_TRIGGER_REF.TimestampFallingEdge:=Ch2_Io_EL1252.TimeStampPos.dwLowPart;
Ch2_XFC_TRIGGER_REF.Edge:=E_SignalEdge.FallingEdge;
Ch2_XFC_TRIGGER_REF.FreeRun:=TRUE;
Ch2_XFC_TRIGGER_REF.ModuloPositions:=FALSE;
Ch2_XFC_TRIGGER_REF.EncoderIndex:=0;//DWORD_TO_UINT(RemAxis.NcToPlc.AxisId);
*)
Ch2_XFC_TRIGGER_REF.Signal:=Ch2_Io_EL1252.Input;
Ch2_XFC_TRIGGER_REF.TimestampRisingEdge:=Ch2_Io_EL1252.TimeStampPos.dwLowPart;
Ch2_XFC_TRIGGER_REF.TimestampFallingEdge:=Ch2_Io_EL1252.TimeStampNeg.dwLowPart;
Ch2_XFC_TRIGGER_REF.Edge:=E_SignalEdge.RisingEdge;
Ch2_XFC_TRIGGER_REF.FreeRun:=TRUE;
Ch2_XFC_TRIGGER_REF.ModuloPositions:=FALSE;
Ch2_XFC_TRIGGER_REF.EncoderIndex:=0;//DWORD_TO_UINT(RemAxis_Ch2.NcToPlc.AxisId);

RemAxis_Ch2.ReadStatus();
Ch2_XFC_TouchProbe(
	Axis:=RemAxis_Ch2 , 
	TriggerInput:=Ch2_XFC_TRIGGER_REF , 
	Execute:=TRUE , 
	WindowOnly:=FALSE , 
	FirstPosition:=0 , 
	LastPosition:=0 , 
	Options:=Ch2_ST_XfcTouchProbeOptions , 
	Done=> , 
	Busy=> , 
	Error=> , 
	ErrorID=> , 
	RecordedPosition=>Ch2_fRecPos );


Ch2_RecTrig(clk:=Ch2_XFC_TouchProbe.Done);
IF EnableOut2 THEN
	IF Ch2_RecTrig.Q THEN
		out2RecPosArray2[Ch2_nRecTimes]:=Ch2_fRecPos;
		Ch2_nRecTimes:=Ch2_nRecTimes+1;
	END_IF
END_IF

Ch2_LogRtrig(clk:=EnableOut2);
IF Ch2_LogRtrig.Q THEN
	FOR Ch2ClearI:=1 TO gMaxPosNum DO
		Out2RecPosArray2[Ch2ClearI]:=0;
	END_FOR
END_IF

Ch2_LogFtrig(clk:=EnableOut2);
IF Ch2_LogFtrig.Q THEN
	Ch2_LogOut:='out2 Pos:,';
	//FOR Ch2_i:=1 TO FlipperOut2Times BY 1 DO
	FOR Ch2_i:=1 TO (Ch2_nRecTimes-1) BY 1 DO
		//Ch2_LogOut:=concat(Ch2_LogOut,LREAL_TO_STRING(out2RecPosArray2[Ch2_i]));
		Ch2_LogOut:=concat(Ch2_LogOut,LREAL_TO_FMTSTR(out2RecPosArray2[Ch2_i],5,FALSE));
		Ch2_LogOut:=concat(Ch2_LogOut,',');
	END_FOR
	Ch2_nRecTimes:=1;
END_IF
END_METHOD

METHOD PRIVATE EL2262
VAR_INPUT
END_VAR
//*******************   output 1  *****************************//
Ch1_ST_CamSwitchOptions.EncoderIndex:=0;//DWORD_TO_UINT(RefAxis.NcToPlc.AxisId);
Ch1_ST_CamSwitchOptions.UseAcceleration:=TRUE;//FALSE TRUE

Ch1_TRACK_REF.ModuloPositions:=FALSE;//启用 模位置
Ch1_TRACK_REF.Disable:=FALSE;
Ch1_TRACK_REF.Force:=ForceOut1;
Ch1_TRACK_REF.OnCompensation:=0;//延时 ON
Ch1_TRACK_REF.OffCompensation:=0;//延时 OFF

RefAxis_Ch1.ReadStatus();
Ch1_MC_DigitalCamSwitch(
	Axis:=RefAxis_Ch1 , 
	Switches:=Ch1_CAMSWITCH_REF , 
	Output:=Ch1_OUTPUT_REF , 
	TrackOptions:=Ch1_TRACK_REF , 
	Enable:=EnableOut1 , 
	Options:=Ch1_ST_CamSwitchOptions , 
	InOperation=> , 
	Busy=> , 
	Error=> , 
	ErrorID=> );
(*
IF RefAxis_Ch1.Status.NotMoving THEN
	Ch1_MC_DigitalCamSwitch(
		Axis:=RefAxis_Ch1 , 
		Switches:=Ch1_CAMSWITCH_REF , 
		Output:=Ch1_OUTPUT_REF , 
		TrackOptions:=Ch1_TRACK_REF , 
		Enable:=FALSE , 
		Options:=Ch1_ST_CamSwitchOptions , 
		InOperation=> , 
		Busy=> , 
		Error=> , 
		ErrorID=> );
END_IF
*)
//*******************   output 2  *****************************//
Ch2_ST_CamSwitchOptions.EncoderIndex:=0;//DWORD_TO_UINT(RefAxis.NcToPlc.AxisId);
Ch2_ST_CamSwitchOptions.UseAcceleration:=TRUE;//FALSE TRUE

Ch2_TRACK_REF.ModuloPositions:=FALSE;//启用 模位置
Ch2_TRACK_REF.Disable:=FALSE;
Ch2_TRACK_REF.Force:=ForceOut2;
Ch2_TRACK_REF.OnCompensation:=0;//延时 ON
Ch2_TRACK_REF.OffCompensation:=0;//延时 OFF

RefAxis_Ch2.ReadStatus();
Ch2_MC_DigitalCamSwitch(
	Axis:=RefAxis_Ch2 , 
	Switches:=Ch2_CAMSWITCH_REF , 
	Output:=Ch2_OUTPUT_REF , 
	TrackOptions:=Ch2_TRACK_REF , 
	Enable:=EnableOut2 , 
	Options:=Ch2_ST_CamSwitchOptions , 
	InOperation=> , 
	Busy=> , 
	Error=> , 
	ErrorID=> );
(*
IF RefAxis_Ch2.Status.NotMoving THEN
	Ch2_MC_DigitalCamSwitch(
		Axis:=RefAxis_Ch2 , 
		Switches:=Ch2_CAMSWITCH_REF , 
		Output:=Ch2_OUTPUT_REF , 
		TrackOptions:=Ch2_TRACK_REF , 
		Enable:=FALSE , 
		Options:=Ch2_ST_CamSwitchOptions , 
		InOperation=> , 
		Busy=> , 
		Error=> , 
		ErrorID=> );
END_IF
*)
//***************** EL2262 *****************************//
Flipper_CH1_XFC_EL2262(
	OversamplingFactor:= OversamplingFactor, 
	OutputOneCycleDelayed:= FALSE, 
	ForceWhenLate:= TRUE, 
	Channel:= 0, 
	Error=> , 
	ErrorID=> , 
	ErrorOutputMissed=> , 
	PrecisionReduced=> , 
	Output:= Ch1_OUTPUT_REF, 
	TrackOptions:= Ch1_TRACK_REF, 
	EL2262:= Io_EL2262);

Flipper_CH2_XFC_EL2262(
	OversamplingFactor:= OversamplingFactor, 
	OutputOneCycleDelayed:= FALSE, 
	ForceWhenLate:= TRUE, 
	Channel:= 1, 
	Error=> , 
	ErrorID=> , 
	ErrorOutputMissed=> , 
	PrecisionReduced=> , 
	Output:= Ch2_OUTPUT_REF, 
	TrackOptions:= Ch2_TRACK_REF, 
	EL2262:= Io_EL2262_Ch2);
END_METHOD

ACTION VersionLog:
(*
版本: V1.0.0.0
说明:
	1. 首个版本
/**************************************************/
版本: V1.0.0.1
说明:
	1. 增加触发上升沿清空EL1252位置记录数据
/**************************************************/
*)
END_ACTION

END_FUNCTION_BLOCK

// ---- POUs/BaseModule/EL2252_2262Control/SquareWaveOut/FB_SquareWaveOut_EL2262.TcPOU
FUNCTION_BLOCK FB_SquareWaveOut_EL2262
VAR_INPUT
	bStart_ch1:BOOL;
	nCycle_ch1:UDINT;//方波周期，需要设置为2的整数倍；单位us
	bStart_ch2:BOOL;
	nCycle_ch2:UDINT;//方波周期，需要设置为2的整数倍；单位us
END_VAR
VAR_OUTPUT
	Io_EL2262:ST_EL2262OutData;//硬件IO，需要关联至EL2262
END_VAR
VAR
	bInitValue1:BOOL;
	nInitCount1:UDINT;
	bInitValue2:BOOL;
	nInitCount2:UDINT;
	i_Temp:INT;
END_VAR

IF bStart_ch1 AND nCycle_ch1>0 THEN
	SetChannelData_Single(OutData:=Io_EL2262.Output0,bInitValue:=bInitValue1,nInitCount:=nInitCount1,nCycle:=nCycle_ch1);
ELSE
	FOR i_Temp:=0 TO 124 DO
		Io_EL2262.Output0[i_Temp]:=0;
	END_FOR
	bInitValue1:=FALSE;
	nInitCount1:=0;
END_IF
IF bStart_ch2 AND nCycle_ch2>0 THEN
	SetChannelData_Single(OutData:=Io_EL2262.Output1,bInitValue:=bInitValue2,nInitCount:=nInitCount2,nCycle:=nCycle_ch2);
ELSE
	FOR i_Temp:=0 TO 124 DO
		Io_EL2262.Output1[i_Temp]:=0;
	END_FOR
	bInitValue2:=FALSE;
	nInitCount2:=0;
END_IF

METHOD Act_Ex_Ch1 : BOOL
VAR_INPUT
END_VAR
IF nCycle_ch1>0 THEN
	bStart_ch1:=TRUE;
	Act_Ex_Ch1:=TRUE;
ELSE
	Act_Ex_Ch1:=FALSE;
END_IF
END_METHOD

METHOD Act_Ex_Ch2 : BOOL
VAR_INPUT
END_VAR
IF nCycle_ch2>0 THEN
	bStart_ch2:=TRUE;
	Act_Ex_Ch2:=TRUE;
ELSE
	Act_Ex_Ch2:=FALSE;
END_IF
END_METHOD

METHOD Act_Stop_Ch1 : BOOL
VAR_INPUT
END_VAR
bStart_ch1:=FALSE;
Act_Stop_Ch1:=TRUE;
END_METHOD

METHOD Act_Stop_Ch2 : BOOL
VAR_INPUT
END_VAR
bStart_ch2:=FALSE;
Act_Stop_Ch2:=TRUE;
END_METHOD

METHOD PRIVATE SetChannelData_Single
VAR_IN_OUT
	OutData							:ARRAY[0..124] OF BYTE;
	bInitValue						:BOOL;
	nInitCount						:UDINT;
END_VAR
VAR_INPUT
	nCycle							:UDINT;//方波周期，建议设置为2的整数倍；单位us, 最大值1000us
END_VAR
VAR
	nPulsWidth						:UDINT;
	i_Byte							:UDINT;
	nByte							:UDINT;
	i_Temp							:UDINT;
	i_Temp1							:UDINT;
	i_Count							:UDINT;
	b_Temp							:BOOL;
END_VAR
//计算电平脉宽
IF nCycle<2 THEN
	nPulsWidth:=1;
ELSE
	nPulsWidth:=nCycle/2;
END_IF

IF nInitCount<=0 THEN
	i_Temp1:=0;
ELSIF nInitCount<1000 THEN
	FOR i_Temp:=0 TO nInitCount BY 1 DO
		IF i_Temp>=8 THEN
			i_Byte:=i_Temp/8;
			nByte:=i_Temp MOD 8;
		ELSE
			i_Byte:=0;
			nByte:=i_Temp;
		END_IF
		CASE nByte OF
			0:
				OutData[i_Byte].0:=bInitValue;
			1:
				OutData[i_Byte].1:=bInitValue;
			2:
				OutData[i_Byte].2:=bInitValue;
			3:
				OutData[i_Byte].3:=bInitValue;
			4:
				OutData[i_Byte].4:=bInitValue;
			5:
				OutData[i_Byte].5:=bInitValue;
			6:
				OutData[i_Byte].6:=bInitValue;
			7:
				OutData[i_Byte].7:=bInitValue;
		END_CASE
	END_FOR
	i_Temp1:=i_Temp;
	bInitValue:=NOT bInitValue;//状态取反
ELSE
	IF bInitValue THEN
		FOR i_Temp:=0 TO 124 DO
			OutData[i_Temp]:=255;
		END_FOR
	ELSE
		FOR i_Temp:=0 TO 124 DO
			OutData[i_Temp]:=0;
		END_FOR
	END_IF
	nInitCount:=nInitCount-1000;//计算剩余值
	IF nInitCount=0 THEN
		bInitValue:=NOT bInitValue;//状态取反
	END_IF
	RETURN;
END_IF
nInitCount:=0;//清空剩余值

//
i_Count:=1;
FOR i_Temp:=i_Temp1 TO 999 BY 1 DO
	IF i_Temp>=8 THEN
		i_Byte:=i_Temp/8;
		nByte:=i_Temp MOD 8;
	ELSE
		i_Byte:=0;
		nByte:=i_Temp;
	END_IF
	CASE nByte OF
		0:
			OutData[i_Byte].0:=bInitValue;
		1:
			OutData[i_Byte].1:=bInitValue;
		2:
			OutData[i_Byte].2:=bInitValue;
		3:
			OutData[i_Byte].3:=bInitValue;
		4:
			OutData[i_Byte].4:=bInitValue;
		5:
			OutData[i_Byte].5:=bInitValue;
		6:
			OutData[i_Byte].6:=bInitValue;
		7:
			OutData[i_Byte].7:=bInitValue;
	END_CASE
	i_Count:=i_Count+1;
	IF i_Count>nPulsWidth THEN
		i_Count:=1;
		bInitValue:=NOT bInitValue;
	END_IF
END_FOR
IF i_Count>1 THEN
	nInitCount:=nPulsWidth-i_Count+1;//计算剩余值
END_IF
//nInitCount:=nPulsWidth-(1000 MOD nPulsWidth);//计算剩余值



(*
//初始化输出，全部置位为高电平
nByte:=125;
FOR i_Byte:=0 TO (nByte-1) DO
	OutData[i_Byte]:=255;
END_FOR

//计算电平脉宽
nPulsWidth:=nCycle/2;

//
i_Count:=1;
b_Temp:=FALSE;
FOR i_Temp:=1 TO 1000 BY 1 DO
	IF i_Temp>8 THEN
		i_Byte:=i_Temp/8;
		nByte:=(i_Temp MOD 8)-1;
	ELSE
		i_Byte:=0;
		nByte:=i_Temp-1;
	END_IF
	IF NOT b_Temp AND i_Count<=nPulsWidth THEN
		CASE nByte OF
			0:
				OutData[i_Byte].0:=0;
			1:
				OutData[i_Byte].1:=0;
			2:
				OutData[i_Byte].2:=0;
			3:
				OutData[i_Byte].3:=0;
			4:
				OutData[i_Byte].4:=0;
			5:
				OutData[i_Byte].5:=0;
			6:
				OutData[i_Byte].6:=0;
			7:
				OutData[i_Byte].7:=0;
		END_CASE
	END_IF
	i_Count:=i_Count+1;
	IF i_Count>nPulsWidth THEN
		i_Count:=1;
		b_Temp:=NOT b_Temp;
	END_IF
END_FOR
*)
END_METHOD

END_FUNCTION_BLOCK

// ---- POUs/BaseModule/EL2252_2262Control/SquareWaveOut/SquareWaveOut_EL2262_TEST.TcPOU
PROGRAM SquareWaveOut_EL2262_TEST
VAR_INPUT
	bStart_ch1:BOOL;
	nCycle_ch1:UDINT;//方波周期，需要设置为2的整数倍；单位us
	bStart_ch2:BOOL;
	nCycle_ch2:UDINT;//方波周期，需要设置为2的整数倍；单位us
END_VAR
VAR
	fb_FB_SquareWaveOut_EL2262:FB_SquareWaveOut_EL2262;
END_VAR


IF bStart_ch1 THEN
	fb_FB_SquareWaveOut_EL2262.Act_Ex_Ch1();
	bStart_ch1:=FALSE;
END_IF
IF bStart_ch2 THEN
	fb_FB_SquareWaveOut_EL2262.Act_Ex_Ch2();
	bStart_ch2:=FALSE;
END_IF
fb_FB_SquareWaveOut_EL2262(
	bStart_ch1:= , 
	nCycle_ch1:= nCycle_ch1, 
	bStart_ch2:= , 
	nCycle_ch2:= nCycle_ch2, 
	Io_EL2262=> );

METHOD Act_Ex_Ch1 : BOOL
VAR_INPUT
END_VAR
Act_Ex_Ch1:=fb_FB_SquareWaveOut_EL2262.Act_Ex_Ch1();
END_METHOD

METHOD Act_Ex_Ch2 : BOOL
VAR_INPUT
END_VAR
Act_Ex_Ch2:=fb_FB_SquareWaveOut_EL2262.Act_Ex_Ch2();
END_METHOD

METHOD Act_Stop_Ch1 : BOOL
VAR_INPUT
END_VAR
bStart_ch1:=FALSE;
Act_Stop_Ch1:=TRUE;
END_METHOD

METHOD Act_Stop_Ch2 : BOOL
VAR_INPUT
END_VAR
bStart_ch2:=FALSE;
Act_Stop_Ch2:=TRUE;
END_METHOD

END_PROGRAM

// ---- POUs/BaseModule/Error/ErrCodeProcess.TcPOU
FUNCTION ErrCodeProcess : LINT
VAR_INPUT
	errorID					:DINT;//error id
END_VAR
VAR
	machineNum:INT;
	levelNum:INT;
	stationNum:INT;
	
	cal_Temp:LINT;
END_VAR

machineNum:=1;
CASE gErrorARRAY[errorID].eErrLevel OF
	Error_Level_0:
		levelNum:=0;
	Error_Level_1:
		levelNum:=1;
	Error_Level_2:
		levelNum:=2;
	Error_Level_3:
		levelNum:=3;
	Error_Level_4:
		levelNum:=4;
END_CASE

IF 0<=errorID AND errorID<=999 THEN// 整机
	stationNum:=0;
	cal_Temp:=machineNum*1000000+stationNum*10000+levelNum*1000+(errorID-0);// 1003000~1003999
ELSIF 1000<=errorID AND errorID<=1999 THEN// 工站1
	stationNum:=1;
	cal_Temp:=machineNum*1000000+stationNum*10000+levelNum*1000+(errorID-1000);// 1013000~1013999
ELSIF 2000<=errorID AND errorID<=2999 THEN// 工站2
	stationNum:=2;
	cal_Temp:=machineNum*1000000+stationNum*10000+levelNum*1000+(errorID-2000);// 1023000~1023999
ELSIF 3000<=errorID AND errorID<=3999 THEN// 工站3
	stationNum:=3;
	cal_Temp:=machineNum*1000000+stationNum*10000+levelNum*1000+(errorID-3000);// 1033000~1033999
ELSIF 4000<=errorID AND errorID<=4999 THEN// 工站4
	stationNum:=4;
	cal_Temp:=machineNum*1000000+stationNum*10000+levelNum*1000+(errorID-4000);// 1043000~1043999
ELSIF 6000<=errorID AND errorID<=6999 THEN// 上料
	stationNum:=6;
	cal_Temp:=machineNum*1000000+stationNum*10000+levelNum*1000+(errorID-6000);// 1063000~1063999
ELSIF 7000<=errorID AND errorID<=7999 THEN// 下料
	stationNum:=7;
	cal_Temp:=machineNum*1000000+stationNum*10000+levelNum*1000+(errorID-7000);// 1073000~1073999
ELSE
	cal_Temp:=0;
END_IF

ErrCodeProcess:=cal_Temp;

END_FUNCTION

// ---- POUs/BaseModule/IO/ReadWriteCSV/POU_Test.TcPOU
PROGRAM POU_Test
VAR
	readBuff:ARRAY [1..10] OF ST_DataFmtBase;
	fbFileReadWrite:FB_IOFileReadWrite;
END_VAR

fbFileReadWrite(
	readBuff:= readBuff, 
	sFileName:= 'E:\FilePath\file.csv', 
	bRead:= , 
	sTxtHead:= 'GROUP,NUM,ENG,CHN,NO USE', 
	bBusy=> , 
	bDone=> , 
	bError=> , 
	nErrid=> );

END_PROGRAM

// ---- POUs/Communication/Communication_Error.TcPOU
PROGRAM Communication_Error
VAR
	f_SWconnect:F_TRIG;

	f_CCDSW1connect:F_TRIG;
	f_CCDSW2connect:F_TRIG;
	f_CCDSW3connect:F_TRIG;
	f_CCDSW4connect:F_TRIG;
	f_CCDSW5connect:F_TRIG;
	f_CCDSW6connect:F_TRIG;
	f_CCDSW7connect:F_TRIG;
	f_CCDSW8connect:F_TRIG;
	f_CCDSW9connect:F_TRIG;
	f_CCDSW10connect:F_TRIG;
	f_CCDSW11connect:F_TRIG;
	f_LocalWconnect:F_TRIG;
	
	
	
	choosedelayTime1:TON;
	choosedelayTime2:TON;
	choosedelayTime3:TON;
	choosedelayTime4:TON;
	choosedelayTime5:TON;
	choosedelayTime6:TON;
	choosedelayTime7:TON;
	choosedelayTime8:TON;
	choosedelayTime9:TON;
	choosedelayTime10:TON;
	choosedelayTime11:TON;
	choosedelayTime12:TON;
	choosedelayTime13:TON;
	
	choosedelayTime14:TON;
	choosedelayTime15:TON;
	choosedelayTime16:TON;
	
	delayTime:TIME:=T#5S;
	
	gEnaConnectRTrig:R_Trig;
	gEnaConnectFTrig:F_Trig;
END_VAR


choosedelayTime1(IN:=gEnableSWConnect , PT:= delayTime, Q=> , ET=> );
choosedelayTime2(IN:=gEnableSWConnect , PT:= delayTime, Q=> , ET=> );



IF (NOT gSWConnected AND choosedelayTime1.Q) THEN
	error_Trigger(91);//主站 上位机通讯断开
END_IF
IF (NOT gSWConnected AND choosedelayTime2.Q) THEN
	error_Trigger(96);//LCCD1 上位机通讯断开
END_IF




/////////////////


f_SWconnect(CLK:=gSWConnected);
f_CCDSW1connect(CLK:=gSWStringConnected);

IF f_SWconnect.Q THEN
	error_Trigger(91);// 主站 软件断开连接
END_IF
IF f_CCDSW1connect.Q THEN
	error_Trigger(96);// 
END_IF
//IF (gCtrlMode=1 OR gAutoRunningFlag) THEN//自动过程中，软件掉线，是否需要重启？
//	IF f_SWconnect.Q OR f_CCDSW1connect.Q THEN
//		gSWDisconnected:=TRUE;
//	END_IF
//END_IF


gEnaConnectRTrig(CLK:=gEnableSWConnectAll , Q=> );
gEnaConnectFTrig(CLK:=gEnableSWConnectAll, Q=> );

//所有软件连接
IF gEnaConnectRTrig.Q THEN
	gEnableSWConnect:=TRUE;
END_IF
//所有软件断开连接
IF gEnaConnectFTrig.Q THEN
	gEnableSWConnect:=FALSE;
END_IF

END_PROGRAM

// ---- POUs/Communication/PLC_FreeByte.TcPOU
PROGRAM PLC_FreeByte
VAR_INPUT
	nSocketType:UINT:=0;// socket 类型; 0 表示 server; 1 表示 client;
	sTerminalName:STRING;// 通讯对方名称 自定义
	sHost:STRING(20):='127.0.0.1';// 通讯IP地址; server时表示本地host; client时表示远程host
	nPort:UDINT:=8900;// 通讯端口号;
	bEnable:BOOL:=TRUE;// 通讯启用\禁用连接
	sSendSuffix:STRING:='';//此处可统一添加发送后缀字符 $R$N
	nQueueInterval:UDINT:=50;// 发送队列时间间隔 单位ms
	logHandleArray:ARRAY [1..5] OF POINTER TO printLogModule_EX;// log 操作 handle 数组
	logHandleArrayLength:UINT:=0;// log 操作 handle 数组长度, 不超过5
END_VAR
VAR_OUTPUT
	bSendCondition	:BOOL;//可发送条件
	bSocketConnected:BOOL;//连接状态
END_VAR
VAR CONSTANT
	cNumBegin		:DINT:=1;
	cNumEnd			:DINT:=100;
END_VAR
VAR
	sendDataArray	:ARRAY [cNumBegin..cNumEnd] OF struct_byte;
	length			:DINT:=0;
	endPoint		:DINT:=cNumBegin;
	popupSendData	:struct_byte;
	//popup
	popupStep		:UINT:=0;
	popupTON1		:TON;
	popupTON2		:TON;
	iPopup			:DINT:=0;
	_PopupLength	:DINT:=0;
END_VAR
VAR
	tcpipClient					:tcpipClientModule_EX;
	tcpipServer					:tcpipServerModule_EX;////定义服务器对象
	
	tcpipSendDataBuff_Server	:struct_byte;//发送数据 Buff server
	tcpipSendDataBuff_Client	:struct_byte;//发送数据 Buff client
	
	tcpipSendDataClear			:struct_byte;//发送数据 清空
	tcpipSendData				:struct_byte;//发送数据
	
	tcpipRecDataBuff_Server		:struct_byte;//已接收数据 Buff server
	tcpipRecDataBuff_Client		:struct_byte;//已接收数据 Buff client
	
	tcpipRecDataClear			:struct_byte;//已接收数据 清空
	tcpipRecData				:struct_byte;//已接收数据
	
	tcpConnectR_Trig			:R_Trig;//初始连接上升沿
	tcpConnectF_Trig			:F_Trig;//初始连接下降沿
	registerStep				:UDINT;//ALC注册控制步
	registerTON					:TON;//ALC注册延时
	
	logHandleArray_index		:UINT:=1;
END_VAR
VAR
	bTrig_Start:BOOL;
	rTrig_Start:R_TRIG;
	tTrig_Start:TON;
	
	bTrig_Stop:BOOL;
	rTrig_Stop:R_TRIG;
	tTrig_Stop:TON;
	
	bTrig_Reset:BOOL;
	rTrig_Reset:R_TRIG;
	tTrig_Reset:TON;
	
	
	bTrig_Init:BOOL;
	rTrig_Init:R_TRIG;
	
	bTrig_All_Home:BOOL;
	rTrig_All_Home:R_TRIG;
	
	bTrig_Z_Safe:BOOL;
	rTrig_Z_Safe:R_TRIG;
	
	bTrig_P_Pos_:BOOL;
	rTrig_P_Pos_:R_TRIG;
	nTrig_P_Pos_TrayNum:UINT:=1;
	nTrig_P_Pos_RowNum:UINT:=1;
	
	bTrig_Move_P_:BOOL;
	rTrig_Move_P_:R_TRIG;
	nTrig_Move_P_TrayNum:UINT:=1;
	nTrig_Move_P_RowNum:UINT:=1;
	nTrig_Move_P_PosNum:UINT:=1;
	findposstart	:INT;
	findposend		:INT;
	find_pos		:INT;
	recStrTemp		:struct_byte;
END_VAR


CASE nSocketType OF
0://TCPIP server
	tcpipServer(
		sSrvNetId:= , 
		sLocalHost:=sHost , 
		nLocalPort:=nPort , 
		bStartConnect:=bEnable , 
		tcpipSDataLen:=20 , 
		tcpipSData:=ADR(tcpipSendDataBuff_Server) , 
		bSend:= , 
		tcpipRecDataLen:=SIZEOF(tcpipRecDataBuff_Server) , 
		tcpipRecData:=ADR(tcpipRecDataBuff_Server) , 
		bAccepted=> , 
		bSendBusy=> , 
		bRecData=> );
	bSendCondition:=tcpipServer.bAccepted AND NOT tcpipServer.bSendBusy;
	//TCPIP连接
	bSocketConnected:=tcpipServer.bAccepted;
	IF NOT tcpipServer.bAccepted THEN
		length:=0;
		endPoint:=cNumBegin;
	END_IF
	tcpConnectR_Trig(CLK:=tcpipServer.bAccepted);
	tcpConnectF_Trig(CLK:=tcpipServer.bAccepted);

1://TCPIP client
	tcpipClient(
		sSrvNetId:= , 
		sRemoteHost:=sHost , 
		nRemotePort:=nPort , 
		bStartConnect:=bEnable , 
		tcpipSDataLen:=20, 
		tcpipSData:=ADR(tcpipSendDataBuff_Client) , 
		bSend:= , 
		tcpipRecDataLen:=SIZEOF(tcpipRecDataBuff_Client) , 
		tcpipRecData:=ADR(tcpipRecDataBuff_Client) , 
		bConnected=> , 
		bSendBusy=> , 
		bRecData=> );
	bSendCondition:=tcpipClient.bConnected AND NOT tcpipClient.bSendBusy;
	//TCPIP连接
	bSocketConnected:=tcpipClient.bConnected;
	IF NOT tcpipClient.bConnected THEN
		length:=0;
		endPoint:=cNumBegin;
	END_IF
	tcpConnectR_Trig(CLK:=tcpipClient.bConnected);
	tcpConnectF_Trig(CLK:=tcpipClient.bConnected);
END_CASE

IF tcpConnectR_Trig.Q THEN
	FOR logHandleArray_index:=1 TO logHandleArrayLength DO
		logHandleArray[logHandleArray_index]^.append(CONCAT(sTerminalName, ' has been connected'));
	END_FOR
	registerStep:=10;
END_IF
IF tcpConnectF_Trig.Q THEN
	FOR logHandleArray_index:=1 TO logHandleArrayLength DO
		logHandleArray[logHandleArray_index]^.append(CONCAT(sTerminalName, ' has been disconnected'));
	END_FOR
	registerStep:=0;
END_IF
//数据接收处理
CASE nSocketType OF
0://TCPIP server
	IF tcpipServer.bRecData THEN
		tcpipRecData:=tcpipRecDataBuff_Server;//buff转存
		tcpipRecDataBuff_Server:=tcpipRecDataClear;//转存之后清空buff
		dataProcessing();
	END_IF
1://TCPIP client
	IF tcpipClient.bRecData THEN
		tcpipRecData:=tcpipRecDataBuff_Client;//buff转存
		tcpipRecDataBuff_Client:=tcpipRecDataClear;//转存之后清空buff
		dataProcessing();
	END_IF
END_CASE


popup();

CASE registerStep OF
0:
	//Ready
END_CASE

ACTION ACT_dataProcessing_DOE:
//(*LoadCCD3*)
//	recStrFilArrSocket[1]:='CoaxialCCD1:';
//	recStrFilArrSocket[2]:='DUTTopX:';
//	recStrFilArrSocket[3]:='DUTTopY:';
//	recStrFilArrSocket[4]:='DUTBottomX:';
//	recStrFilArrSocket[5]:='DUTBottomY:';
//	recStrFilArrSocket[6]:='SocketTopX:';
//	recStrFilArrSocket[7]:='SocketTopY:';
//	recStrFilArrSocket[8]:='SocketBottomX:';
//	recStrFilArrSocket[9]:='SocketBottomY:';
//	recStrFilArrSocket[10]:='ModelAngle:';
	
//	recStrTemp:='';
//	find_pos:=FIND(tcpipRecData, recStrFilArrSocket[1]);
//	IF find_pos>0 THEN
//		findposstart:=find_pos;
//		find_pos:=0;
//		find_pos:=FIND(tcpipRecData, ';');
//		IF find_pos>0 THEN
//			findposend:=find_pos;
//			find_pos:=0;
//		END_IF
//		recPosArrSocket_G_CCD1[1]:=STRING_TO_LREAL(MID(tcpipRecData,findposend-findposstart-(len(recStrFilArrSocket[1])+len(recStrFilArrSocket[2])),findposstart+len(recStrFilArrSocket[1])+len(recStrFilArrSocket[2])));
//		recStrTemp:=DELETE(tcpipRecData,findposend-findposstart+1,findposstart);
//		find_pos:=0;
//		findposstart:=1;
//		find_pos:=FIND(recStrTemp, ';');
//		IF find_pos>0 THEN
//			findposend:=find_pos;
//			find_pos:=0;
//		END_IF
//		recPosArrSocket_G_CCD1[2]:=STRING_TO_LREAL(MID(recStrTemp,findposend-findposstart-len(recStrFilArrSocket[3]),findposstart+len(recStrFilArrSocket[3])));
//		recStrTemp:=DELETE(recStrTemp,findposend-findposstart+1,findposstart);
//		find_pos:=0;
//		findposstart:=1;
//		find_pos:=FIND(recStrTemp, ';');
//		IF find_pos>0 THEN
//			findposend:=find_pos;
//			find_pos:=0;
//		END_IF
//		recPosArrSocket_G_CCD1[3]:=STRING_TO_LREAL(MID(recStrTemp,findposend-findposstart-len(recStrFilArrSocket[4]),findposstart+len(recStrFilArrSocket[4])));
//		recStrTemp:=DELETE(recStrTemp,findposend-findposstart+1,findposstart);
//		find_pos:=0;
//		findposstart:=1;
//		find_pos:=FIND(recStrTemp, ';');
//		IF find_pos>0 THEN
//			findposend:=find_pos;
//			find_pos:=0;
//		END_IF
//		recPosArrSocket_G_CCD1[4]:=STRING_TO_LREAL(MID(recStrTemp,findposend-findposstart-len(recStrFilArrSocket[5]),findposstart+len(recStrFilArrSocket[5])));
//		recStrTemp:=DELETE(recStrTemp,findposend-findposstart+1,findposstart);
//		find_pos:=0;
//		findposstart:=1;
//		find_pos:=FIND(recStrTemp, ';');
//		IF find_pos>0 THEN
//			findposend:=find_pos;
//			find_pos:=0;
//		END_IF
//		recPosArrSocket_G_CCD1[5]:=STRING_TO_LREAL(MID(recStrTemp,findposend-findposstart-len(recStrFilArrSocket[6]),findposstart+len(recStrFilArrSocket[6])));
//		recStrTemp:=DELETE(recStrTemp,findposend-findposstart+1,findposstart);
//		find_pos:=0;
//		findposstart:=1;
//		find_pos:=FIND(recStrTemp, ';');
//		IF find_pos>0 THEN
//			findposend:=find_pos;
//			find_pos:=0;
//		END_IF
//		recPosArrSocket_G_CCD1[6]:=STRING_TO_LREAL(MID(recStrTemp,findposend-findposstart-len(recStrFilArrSocket[7]),findposstart+len(recStrFilArrSocket[7])));
//		recStrTemp:=DELETE(recStrTemp,findposend-findposstart+1,findposstart);
//		find_pos:=0;
//		findposstart:=1;
//		find_pos:=FIND(recStrTemp, ';');
//		IF find_pos>0 THEN
//			findposend:=find_pos;
//			find_pos:=0;
//		END_IF
//		recPosArrSocket_G_CCD1[7]:=STRING_TO_LREAL(MID(recStrTemp,findposend-findposstart-len(recStrFilArrSocket[8]),findposstart+len(recStrFilArrSocket[8])));
//		recStrTemp:=DELETE(recStrTemp,findposend-findposstart+1,findposstart);
//		find_pos:=0;
//		findposstart:=1;
//		find_pos:=FIND(recStrTemp, ';');
//		IF find_pos>0 THEN
//			findposend:=find_pos;
//			find_pos:=0;
//		END_IF
//		recPosArrSocket_G_CCD1[8]:=STRING_TO_LREAL(MID(recStrTemp,findposend-findposstart-len(recStrFilArrSocket[9]),findposstart+len(recStrFilArrSocket[9])));
//		recStrTemp:=DELETE(recStrTemp,findposend-findposstart+1,findposstart);
//		find_pos:=0;
//		findposstart:=1;
//		find_pos:=FIND(recStrTemp, ';');
//		IF find_pos>0 THEN
//			findposend:=find_pos;
//			find_pos:=0;
//		END_IF
//		recPosArrSocket_G_CCD1[9]:=STRING_TO_LREAL(MID(recStrTemp,findposend-findposstart-len(recStrFilArrSocket[10]),findposstart+len(recStrFilArrSocket[10])));
//		recStrTemp:=DELETE(recStrTemp,findposend-findposstart+1,findposstart);
//		recCCDResultArr[3]:=TRUE;
//	END_IF
END_ACTION

METHOD appendSend : BOOL
VAR_INPUT
	str			:struct_byte;
END_VAR
VAR
	suffix					:struct_byte;
	strTemp_appendSend		:struct_byte;
END_VAR

IF endPoint>(cNumEnd-1) THEN
	RETURN;
END_IF

strTemp_appendSend:=str;
sendDataArray[endPoint]:=strTemp_appendSend;

endPoint:=endPoint+1;
length:=endPoint-cNumBegin;
END_METHOD

METHOD dataProcessing : BOOL
VAR_INPUT
END_VAR
VAR
	str1:STRING;
END_VAR
FOR logHandleArray_index:=1 TO logHandleArrayLength DO
	CASE nSocketType OF
	0://TCPIP server
		str1:=CONCAT(str1,BYTE_TO_HEXSTR(tcpipRecData.b1,2,FALSE));
		str1:=CONCAT(str1,' ');
		str1:=CONCAT(str1,BYTE_TO_HEXSTR(tcpipRecData.b2,2,FALSE));
		str1:=CONCAT(str1,' ');
		str1:=CONCAT(str1,BYTE_TO_HEXSTR(tcpipRecData.b3,2,FALSE));
		str1:=CONCAT(str1,' ');
		str1:=CONCAT(str1,BYTE_TO_HEXSTR(tcpipRecData.b4,2,FALSE));
		str1:=CONCAT(str1,' ');
		str1:=CONCAT(str1,BYTE_TO_HEXSTR(tcpipRecData.b5,2,FALSE));
		str1:=CONCAT(str1,' ');
		str1:=CONCAT(str1,BYTE_TO_HEXSTR(tcpipRecData.b6,2,FALSE));
		str1:=CONCAT(str1,' ');
		str1:=CONCAT(str1,BYTE_TO_HEXSTR(tcpipRecData.b7,2,FALSE));
		str1:=CONCAT(str1,' ');
		str1:=CONCAT(str1,BYTE_TO_HEXSTR(tcpipRecData.b8,2,FALSE));
		str1:=CONCAT(str1,' ');
		str1:=CONCAT(str1,BYTE_TO_HEXSTR(tcpipRecData.b9,2,FALSE));
		str1:=CONCAT(str1,' ');
		str1:=CONCAT(str1,BYTE_TO_HEXSTR(tcpipRecData.b10,2,FALSE));
		str1:=CONCAT(str1,' ');
		str1:=CONCAT(str1,BYTE_TO_HEXSTR(tcpipRecData.b11,2,FALSE));
		str1:=CONCAT(str1,' ');
		str1:=CONCAT(str1,BYTE_TO_HEXSTR(tcpipRecData.b12,2,FALSE));
		str1:=CONCAT(str1,' ');
		str1:=CONCAT(str1,BYTE_TO_HEXSTR(tcpipRecData.b13,2,FALSE));
		str1:=CONCAT(str1,' ');
		str1:=CONCAT(str1,BYTE_TO_HEXSTR(tcpipRecData.b14,2,FALSE));
		str1:=CONCAT(str1,' ');
		str1:=CONCAT(str1,BYTE_TO_HEXSTR(tcpipRecData.b15,2,FALSE));
		str1:=CONCAT(str1,' ');
		str1:=CONCAT(str1,BYTE_TO_HEXSTR(tcpipRecData.b16,2,FALSE));
		str1:=CONCAT(str1,' ');
		str1:=CONCAT(str1,BYTE_TO_HEXSTR(tcpipRecData.b17,2,FALSE));
		str1:=CONCAT(str1,' ');
		str1:=CONCAT(str1,BYTE_TO_HEXSTR(tcpipRecData.b18,2,FALSE));
		str1:=CONCAT(str1,' ');
		str1:=CONCAT(str1,BYTE_TO_HEXSTR(tcpipRecData.b19,2,FALSE));
		str1:=CONCAT(str1,' ');
		str1:=CONCAT(str1,BYTE_TO_HEXSTR(tcpipRecData.b20,2,FALSE));
		logHandleArray[logHandleArray_index]^.append(CONCAT(CONCAT(CONCAT('Recevie From ', sTerminalName), ' -- '),str1));
	1://TCPIP client
		str1:=CONCAT(str1,BYTE_TO_HEXSTR(tcpipRecData.b1,2,FALSE));
		str1:=CONCAT(str1,' ');
		str1:=CONCAT(str1,BYTE_TO_HEXSTR(tcpipRecData.b2,2,FALSE));
		str1:=CONCAT(str1,' ');
		str1:=CONCAT(str1,BYTE_TO_HEXSTR(tcpipRecData.b3,2,FALSE));
		str1:=CONCAT(str1,' ');
		str1:=CONCAT(str1,BYTE_TO_HEXSTR(tcpipRecData.b4,2,FALSE));
		str1:=CONCAT(str1,' ');
		str1:=CONCAT(str1,BYTE_TO_HEXSTR(tcpipRecData.b5,2,FALSE));
		str1:=CONCAT(str1,' ');
		str1:=CONCAT(str1,BYTE_TO_HEXSTR(tcpipRecData.b6,2,FALSE));
		str1:=CONCAT(str1,' ');
		str1:=CONCAT(str1,BYTE_TO_HEXSTR(tcpipRecData.b7,2,FALSE));
		str1:=CONCAT(str1,' ');
		str1:=CONCAT(str1,BYTE_TO_HEXSTR(tcpipRecData.b8,2,FALSE));
		str1:=CONCAT(str1,' ');
		str1:=CONCAT(str1,BYTE_TO_HEXSTR(tcpipRecData.b9,2,FALSE));
		str1:=CONCAT(str1,' ');
		str1:=CONCAT(str1,BYTE_TO_HEXSTR(tcpipRecData.b10,2,FALSE));
		str1:=CONCAT(str1,' ');
		str1:=CONCAT(str1,BYTE_TO_HEXSTR(tcpipRecData.b11,2,FALSE));
		str1:=CONCAT(str1,' ');
		str1:=CONCAT(str1,BYTE_TO_HEXSTR(tcpipRecData.b12,2,FALSE));
		str1:=CONCAT(str1,' ');
		str1:=CONCAT(str1,BYTE_TO_HEXSTR(tcpipRecData.b13,2,FALSE));
		str1:=CONCAT(str1,' ');
		str1:=CONCAT(str1,BYTE_TO_HEXSTR(tcpipRecData.b14,2,FALSE));
		str1:=CONCAT(str1,' ');
		str1:=CONCAT(str1,BYTE_TO_HEXSTR(tcpipRecData.b15,2,FALSE));
		str1:=CONCAT(str1,' ');
		str1:=CONCAT(str1,BYTE_TO_HEXSTR(tcpipRecData.b16,2,FALSE));
		str1:=CONCAT(str1,' ');
		str1:=CONCAT(str1,BYTE_TO_HEXSTR(tcpipRecData.b17,2,FALSE));
		str1:=CONCAT(str1,' ');
		str1:=CONCAT(str1,BYTE_TO_HEXSTR(tcpipRecData.b18,2,FALSE));
		str1:=CONCAT(str1,' ');
		str1:=CONCAT(str1,BYTE_TO_HEXSTR(tcpipRecData.b19,2,FALSE));
		str1:=CONCAT(str1,' ');
		str1:=CONCAT(str1,BYTE_TO_HEXSTR(tcpipRecData.b20,2,FALSE));
		logHandleArray[logHandleArray_index]^.append(CONCAT(CONCAT(CONCAT('Recevie From ', sTerminalName), ' -- '),str1));
	END_CASE
END_FOR
findposend:=0;
find_pos:=0;
ACT_dataProcessing_DOE();
END_METHOD

METHOD PRIVATE popup : BOOL
VAR_INPUT
END_VAR
CASE popupStep OF
0:
	IF length>0 AND bSendCondition THEN
		_PopupLength:=length;
		popupSendData:=sendDataArray[cNumBegin];
		FOR iPopup:=cNumBegin TO (_PopupLength-1) DO
			sendDataArray[iPopup]:=sendDataArray[iPopup+1];
		END_FOR
		endPoint:=endPoint-1;
		length:=endPoint-cNumBegin;
		sendData(popupSendData);//此处是调用信息发送
		popupStep:=10;
	END_IF
10:
	popupTON2(IN:=NOT popupTON2.Q, PT:=T#2S);
	IF NOT bSendCondition OR popupTON2.Q THEN
		popupTON2(IN:=FALSE);
		popupStep:=11;
	END_IF
11:
	IF bSendCondition THEN
		popupStep:=12;
	END_IF
	popupTON1(IN:=FALSE);
12:
	//popupTON1(IN:=NOT popupTON1.Q,PT:=T#10MS);
	popupTON1(IN:=NOT popupTON1.Q,PT:=TO_TIME(nQueueInterval));
	IF popupTON1.Q THEN
		popupStep:=0;
	END_IF
END_CASE
END_METHOD

METHOD PRIVATE sendData : BOOL
VAR_INPUT
	dataStruct	:struct_byte;
END_VAR
VAR
	str1:STRING;
END_VAR
IF bSendCondition AND bEnable THEN
	tcpipSendData:=dataStruct;
	
	CASE nSocketType OF
	0://TCPIP server
		tcpipSendDataBuff_Server:=tcpipSendData;
		tcpipSendData:=tcpipSendDataClear;	
		tcpipServer.bSend:=TRUE;
	1://TCPIP client
		tcpipSendDataBuff_Client:=tcpipSendData;
		tcpipSendData:=tcpipSendDataClear;	
		tcpipClient.bSend:=TRUE;
	END_CASE
	
	FOR logHandleArray_index:=1 TO logHandleArrayLength DO
		CASE nSocketType OF
		0://TCPIP server
			str1:=CONCAT(str1,BYTE_TO_HEXSTR(tcpipSendDataBuff_Server.b1,2,FALSE));
			str1:=CONCAT(str1,' ');
			str1:=CONCAT(str1,BYTE_TO_HEXSTR(tcpipSendDataBuff_Server.b2,2,FALSE));
			str1:=CONCAT(str1,' ');
			str1:=CONCAT(str1,BYTE_TO_HEXSTR(tcpipSendDataBuff_Server.b3,2,FALSE));
			str1:=CONCAT(str1,' ');
			str1:=CONCAT(str1,BYTE_TO_HEXSTR(tcpipSendDataBuff_Server.b4,2,FALSE));
			str1:=CONCAT(str1,' ');
			str1:=CONCAT(str1,BYTE_TO_HEXSTR(tcpipSendDataBuff_Server.b5,2,FALSE));
			str1:=CONCAT(str1,' ');
			str1:=CONCAT(str1,BYTE_TO_HEXSTR(tcpipSendDataBuff_Server.b6,2,FALSE));
			str1:=CONCAT(str1,' ');
			str1:=CONCAT(str1,BYTE_TO_HEXSTR(tcpipSendDataBuff_Server.b7,2,FALSE));
			str1:=CONCAT(str1,' ');
			str1:=CONCAT(str1,BYTE_TO_HEXSTR(tcpipSendDataBuff_Server.b8,2,FALSE));
			str1:=CONCAT(str1,' ');
			str1:=CONCAT(str1,BYTE_TO_HEXSTR(tcpipSendDataBuff_Server.b9,2,FALSE));
			str1:=CONCAT(str1,' ');
			str1:=CONCAT(str1,BYTE_TO_HEXSTR(tcpipSendDataBuff_Server.b10,2,FALSE));
			str1:=CONCAT(str1,' ');
			str1:=CONCAT(str1,BYTE_TO_HEXSTR(tcpipSendDataBuff_Server.b11,2,FALSE));
			str1:=CONCAT(str1,' ');
			str1:=CONCAT(str1,BYTE_TO_HEXSTR(tcpipSendDataBuff_Server.b12,2,FALSE));
			str1:=CONCAT(str1,' ');
			str1:=CONCAT(str1,BYTE_TO_HEXSTR(tcpipSendDataBuff_Server.b13,2,FALSE));
			str1:=CONCAT(str1,' ');
			str1:=CONCAT(str1,BYTE_TO_HEXSTR(tcpipSendDataBuff_Server.b14,2,FALSE));
			str1:=CONCAT(str1,' ');
			str1:=CONCAT(str1,BYTE_TO_HEXSTR(tcpipSendDataBuff_Server.b15,2,FALSE));
			str1:=CONCAT(str1,' ');
			str1:=CONCAT(str1,BYTE_TO_HEXSTR(tcpipSendDataBuff_Server.b16,2,FALSE));
			str1:=CONCAT(str1,' ');
			str1:=CONCAT(str1,BYTE_TO_HEXSTR(tcpipSendDataBuff_Server.b17,2,FALSE));
			str1:=CONCAT(str1,' ');
			str1:=CONCAT(str1,BYTE_TO_HEXSTR(tcpipSendDataBuff_Server.b18,2,FALSE));
			str1:=CONCAT(str1,' ');
			str1:=CONCAT(str1,BYTE_TO_HEXSTR(tcpipSendDataBuff_Server.b19,2,FALSE));
			str1:=CONCAT(str1,' ');
			str1:=CONCAT(str1,BYTE_TO_HEXSTR(tcpipSendDataBuff_Server.b20,2,FALSE));
			logHandleArray[logHandleArray_index]^.append(CONCAT(CONCAT(CONCAT('Send To ', sTerminalName), ' -- '),str1));
		1://TCPIP client
			str1:=CONCAT(str1,' ');
			str1:=CONCAT(str1,BYTE_TO_HEXSTR(tcpipSendDataBuff_Client.b1,2,FALSE));
			str1:=CONCAT(str1,' ');
			str1:=CONCAT(str1,BYTE_TO_HEXSTR(tcpipSendDataBuff_Client.b2,2,FALSE));
			str1:=CONCAT(str1,' ');
			str1:=CONCAT(str1,BYTE_TO_HEXSTR(tcpipSendDataBuff_Client.b3,2,FALSE));
			str1:=CONCAT(str1,' ');
			str1:=CONCAT(str1,BYTE_TO_HEXSTR(tcpipSendDataBuff_Client.b4,2,FALSE));
			str1:=CONCAT(str1,' ');
			str1:=CONCAT(str1,BYTE_TO_HEXSTR(tcpipSendDataBuff_Client.b5,2,FALSE));
			str1:=CONCAT(str1,' ');
			str1:=CONCAT(str1,BYTE_TO_HEXSTR(tcpipSendDataBuff_Client.b6,2,FALSE));
			str1:=CONCAT(str1,' ');
			str1:=CONCAT(str1,BYTE_TO_HEXSTR(tcpipSendDataBuff_Client.b7,2,FALSE));
			str1:=CONCAT(str1,' ');
			str1:=CONCAT(str1,BYTE_TO_HEXSTR(tcpipSendDataBuff_Client.b8,2,FALSE));
			str1:=CONCAT(str1,' ');
			str1:=CONCAT(str1,BYTE_TO_HEXSTR(tcpipSendDataBuff_Client.b9,2,FALSE));
			str1:=CONCAT(str1,' ');
			str1:=CONCAT(str1,BYTE_TO_HEXSTR(tcpipSendDataBuff_Client.b10,2,FALSE));
			str1:=CONCAT(str1,' ');
			str1:=CONCAT(str1,BYTE_TO_HEXSTR(tcpipSendDataBuff_Client.b11,2,FALSE));
			str1:=CONCAT(str1,' ');
			str1:=CONCAT(str1,BYTE_TO_HEXSTR(tcpipSendDataBuff_Client.b12,2,FALSE));
			str1:=CONCAT(str1,' ');
			str1:=CONCAT(str1,BYTE_TO_HEXSTR(tcpipSendDataBuff_Client.b13,2,FALSE));
			str1:=CONCAT(str1,' ');
			str1:=CONCAT(str1,BYTE_TO_HEXSTR(tcpipSendDataBuff_Client.b14,2,FALSE));
			str1:=CONCAT(str1,' ');
			str1:=CONCAT(str1,BYTE_TO_HEXSTR(tcpipSendDataBuff_Client.b15,2,FALSE));
			str1:=CONCAT(str1,' ');
			str1:=CONCAT(str1,BYTE_TO_HEXSTR(tcpipSendDataBuff_Client.b16,2,FALSE));
			str1:=CONCAT(str1,' ');
			str1:=CONCAT(str1,BYTE_TO_HEXSTR(tcpipSendDataBuff_Client.b17,2,FALSE));
			str1:=CONCAT(str1,' ');
			str1:=CONCAT(str1,BYTE_TO_HEXSTR(tcpipSendDataBuff_Client.b18,2,FALSE));
			str1:=CONCAT(str1,' ');
			str1:=CONCAT(str1,BYTE_TO_HEXSTR(tcpipSendDataBuff_Client.b19,2,FALSE));
			str1:=CONCAT(str1,' ');
			str1:=CONCAT(str1,BYTE_TO_HEXSTR(tcpipSendDataBuff_Client.b20,2,FALSE));
			logHandleArray[logHandleArray_index]^.append(CONCAT(CONCAT(CONCAT('Send To ', sTerminalName), ' -- '),str1));
		END_CASE
	END_FOR
END_IF
END_METHOD

END_PROGRAM

// ---- POUs/Data/Test_FilePOU.TcPOU
PROGRAM Test_FilePOU
VAR
	testMetho:FB_FileGets;
END_VAR

testMetho(
	sNetId:= , 
	hFile:= , 
	bExecute:= , 
	tTimeout:= , 
	bBusy=> , 
	bError=> , 
	nErrId=> , 
	sLine=> , 
	bEOF=> );

END_PROGRAM

// ---- GlobalTextList.TcGTLO
TEXTLIST GlobalTextList
  89 = '                All Show' | Chinese: '               全部' | English: '               ALL Show'
  1821 = '                Part Show' | Chinese: '              总览' | English: '               Part Show'
  718 = ' ICP01   ' | Chinese: 'ICP' | English: 'ICP'
  1341 = '%' | Chinese: '%' | English: '%'
  593 = '%.1f' | Chinese: '%.1f' | English: '%.1f'
  463 = '%.1f %'
  233 = '%.2f' | Chinese: '%.2f' | English: '%.2f'
  532 = '%.3f' | Chinese: '%.3f' | English: '%.3f'
  231 = '%.4f' | Chinese: '%.4f' | English: '%.4f'
  182 = '%d' | Chinese: '%d' | English: '%d'
  264 = '%s' | Chinese: '%s' | English: '%s'
  1790 = '(10)'
  1500 = '(100)'
  1605 = '(200)'
  512 = '(50)'
  1351 = '(500)'
  600 = '1' | Chinese: '1' | English: '1'
  509 = '1\n(N2)'
  609 = '10' | Chinese: '10' | English: '10'
  400 = '11' | Chinese: '11' | English: '11'
  960 = '12' | Chinese: '12' | English: '12'
  961 = '13' | Chinese: '13' | English: '13'
  962 = '14' | Chinese: '14' | English: '14'
  963 = '15' | Chinese: '15' | English: '15'
  964 = '16' | Chinese: '16' | English: '16'
  2411 = '192.168.1.12'
  2489 = '192.168.1.13'
  1159 = '192.168.1.14'
  1635 = '192.168.1.15'
  3262 = '192.168.1.253'
  601 = '2' | Chinese: '2' | English: '2'
  837 = '2\n(CF4)'
  2024 = '20\n(Main)'
  602 = '3' | Chinese: '3' | English: '3'
  3626 = '3\n(CHF3)'
  603 = '4' | Chinese: '4' | English: '4'
  39 = '4\n(SF6)'
  604 = '5' | Chinese: '5' | English: '5'
  1258 = '5\n(O2)'
  2177 = '5110'
  1962 = '5120'
  3714 = '5130'
  357 = '5140'
  3615 = '5200'
  605 = '6' | Chinese: '6' | English: '6'
  611 = '6\n(O2)'
  606 = '7' | Chinese: '7' | English: '7'
  1337 = '7\n(He)'
  607 = '8' | Chinese: '8' | English: '8'
  2488 = '8\n(Ar)'
  608 = '9' | Chinese: '9' | English: '9'
  2062 = '9\n(C4F8)'
  1248 = 'A'
  508 = 'A:Auto Running\nE:Error Running\nH:Homing\nM:Manual Running\nP:Pause Running\nS:Stop Running'
  757 = 'ACC' | Chinese: '加速' | English: 'ACC'
  1604 = 'ACCELERATE' | Chinese: '加速' | English: 'ACCELERATE'
  1434 = 'ACSw' | Chinese: '加速信号' | English: 'ACSw'
  103 = 'Actor Recover' | Chinese: '执行器复位' | English: 'Actor Recover'
  2689 = 'ADD NEW RECIPE' | Chinese: '新增配方' | English: 'ADD NEW RECIPE'
  2063 = 'ADD STEP' | Chinese: '新增步' | English: 'ADD STEP'
  3464 = 'admin' | Chinese: 'admin' | English: 'admin'
  1052 = 'AIM GAUGE' | Chinese: '腔体真空计' | English: 'AIM Gauge'
  1197 = 'ALL' | Chinese: '全部' | English: 'ALL'
  1188 = 'ALL  STOP' | Chinese: '全部停止' | English: 'ALL STOP'
  1647 = 'ALL Clear' | Chinese: '全部清除' | English: 'ALL Clear'
  1634 = 'ALL Set' | Chinese: '全部设置' | English: 'ALL Set'
  492 = 'ALL STOP' | Chinese: '全部停止' | English: 'ALL STOP'
  882 = 'AlmSw' | Chinese: '报警信号' | English: 'AlmSw'
  1796 = 'AMX IP:'
  3635 = 'AMX Port:'
  3264 = 'Ar(500)'
  210 = 'ARM' | Chinese: '机械手' | English: 'ARM'
  238 = 'Axis Status' | Chinese: '轴状态' | English: 'Axis Status'
  2158 = 'BacHe Port:'
  3570 = 'BacHe RF IP:'
  966 = 'Back' | Chinese: 'Back' | English: 'Back'
  1122 = 'BACK OF HELIUM' | Chinese: '背氦' | English: 'BACK OF HELIUM'
  3376 = 'Baise Config：Disable-Dis OR Enable-En' | Chinese: '基础配置：禁用和使能' | English: 'Baise Config：Disable-Dis OR Enable-En'
  4927 = 'BC:%.1fA' | Chinese: 'BC:%.1A' | English: 'BC:%.1A'
  1873 = 'BRACK' | Chinese: '制动' | English: 'BRACK'
  1934 = 'BT:%.1f℃' | Chinese: 'BT:%.1℃' | English: 'BT:%.1℃'
  187 = 'Busy' | Chinese: '运行中' | English: 'Busy'
  3897 = 'BV:%.1frpm' | Chinese: 'BT:%.1fpm' | English: 'BT:%.1fpm'
  590 = 'BW_Limit' | Chinese: 'BW_Limit' | English: 'BW_Limit'
  2787 = 'C4F8(200)'
  5406 = 'C:%.1fA' | Chinese: 'C:%.1A' | English: 'C:%.1A'
  2077 = 'Cancel' | Chinese: '取消' | English: 'Cancel'
  1538 = 'CF4(200)'
  301 = 'CHAMBER' | Chinese: '腔体' | English: 'CHAMBER'
  3502 = 'Chamber' | Chinese: '腔体' | English: 'Chamber'
  1702 = 'Chamber ' | Chinese: '腔体' | English: 'Chamber'
  1370 = 'Chamber ATM state' | Chinese: '腔体大气' | English: 'Chamber ATM state'
  384 = 'Charmber Vent' | Chinese: '腔体破空' | English: 'Chamber Vent'
  1142 = 'CHF3(200)'
  2293 = 'CHILLER' | Chinese: '水冷机' | English: 'CHILLER'
  1594 = 'Chiller Port:'
  2019 = 'Chillerl IP:'
  2457 = 'Chinese' | Chinese: '中文' | English: 'Chinese'
  2889 = 'Clear Changes' | Chinese: '清除' | English: 'Clear Changes'
  438 = 'Clear Info' | Chinese: '清除信息' | English: 'Clear Info'
  1280 = 'CloEN' | Chinese: '启用关闭' | English: 'CloEN'
  2166 = 'CLOSE' | Chinese: '关闭' | English: 'CLOSE'
  2438 = 'Close' | Chinese: '关闭' | English: 'Close'
  295 = 'Config' | Chinese: '配置' | English: 'Config'
  5846 = 'CsCd' | Chinese: 'CsCd' | English: 'CsCd'
  820 = 'Curr Page' | Chinese: '当前页' | English: 'Curr Page'
  1591 = 'CURRENT' | Chinese: '电流' | English: 'CURRENT'
  206 = 'D:%d' | Chinese: 'D:%d' | English: 'D:%d'
  309 = 'Data Change' | Chinese: '数据变更' | English: 'Data Change'
  3129 = 'DC:%.1fA' | Chinese: 'DC:%.1A' | English: 'DC:%.1A'
  1256 = 'DCC' | Chinese: '减速' | English: 'DCC'
  1499 = 'DCSw' | Chinese: 'DCSw' | English: 'DCSw'
  1048 = 'DEC' | Chinese: '减 ' | English: 'DEC'
  1580 = 'DELETE  RECIPE' | Chinese: '删除配方' | English: 'DELETE RECIPE'
  149 = 'DIRECTION' | Chinese: '点动' | English: 'DIRECTION'
  4575 = 'DL:%.1f' | Chinese: 'DL:%.1f' | English: 'DL:%.1f'
  240 = 'Dog_Prox' | Chinese: 'Dog_Prox' | English: 'Dog_Prox'
  188 = 'Done' | Chinese: '完成' | English: 'Done'
  3154 = 'DRY PUM' | Chinese: '干泵' | English: 'DRY PUM'
  2232 = 'DT:%.1f℃' | Chinese: 'DT:%.1f' | English: 'DT:%.1f'
  506 = 'DV:%.1frpm' | Chinese: 'DV:%.1frpm' | English: 'DV:%.1frpm'
  800 = 'editor' | Chinese: '编辑者' | English: 'editor'
  2584 = 'ELE.' | Chinese: '电台' | English: 'ELE.'
  185 = 'Enable' | Chinese: '启用' | English: 'Enable'
  491 = 'ENABLE' | Chinese: '启用' | English: 'ENABLE'
  507 = 'Enable Beep' | Chinese: '启用蜂鸣器' | English: 'Enable Beep'
  430 = 'Enable Save' | Chinese: '启用保存' | English: 'Enable Save'
  2168 = 'English' | Chinese: '英文' | English: 'English'
  186 = 'ErrID' | Chinese: '错误ID' | English: 'ErrID'
  150 = 'Error' | Chinese: '报错' | English: 'Error'
  1837 = 'Error ' | Chinese: '报错' | English: 'Error'
  1284 = 'ErrSw' | Chinese: 'ErrSw' | English: 'ErrSw'
  2629 = 'Etching' | Chinese: '蚀刻' | English: 'Etching'
  1312 = 'ET_T' | Chinese: 'ET_T ' | English: 'ET_T '
  3456 = 'ExtCd' | Chinese: 'ErrCd' | English: 'ErrCd'
  183 = 'ExtEN' | Chinese: 'ExtEN' | English: 'ExtEN'
  181 = 'ExtSw' | Chinese: 'ExtSw' | English: 'ExtSw'
  1053 = 'FAILURE' | Chinese: '报错' | English: 'FAILURE'
  25 = 'FAST\nVALVE' | Chinese: '主抽阀' | English: 'FAST\nPUM'
  1383 = 'FLOW\n(sccm)' | Chinese: '流量\n(sccm)' | English: 'FLOW\n(sccm)'
  1181 = 'FOR. POWER' | Chinese: '反馈功率' | English: 'FOR. POWER'
  3145 = 'Force Back Of Helium IN Control' | Chinese: '强制背氦进气控制' | English: 'Force Back Of Helium IN Control'
  3586 = 'Force GateDoor Control' | Chinese: '强制GD控制' | English: 'Force GateDoor Control'
  2030 = 'Force PDV Control' | Chinese: '强制PDV控制' | English: 'Force PDV Control'
  847 = 'FORELINE' | Chinese: '前置阀' | English: 'FORELINE'
  589 = 'FW_Limit' | Chinese: 'FW_Limit' | English: 'FW_Limit'
  1140 = 'GAS\nLINE' | Chinese: '气路' | English: 'GAS\nLINE'
  661 = 'GAS BOX' | Chinese: '气柜' | English: 'GAS BOX'
  1836 = 'GAS LINE' | Chinese: '气路' | English: 'GAS LINE'
  683 = 'GATE DOOR' | Chinese: '闸门' | English: 'GATE DOOR'
  2792 = 'Gate Door' | Chinese: '闸门' | English: 'Gate Door'
  804 = 'Go' | Chinese: '执行' | English: 'Go'
  1599 = 'GVA' | Chinese: '前端阀' | English: 'GVA'
  2627 = 'GVA ALL CL' | Chinese: 'GVA 全关' | English: 'GVA ALL CL'
  2227 = 'GVA ALL OP' | Chinese: 'GVA 全开' | English: 'GVA ALL OP'
  1078 = 'GVA10\n(Vent)'
  621 = 'GVB' | Chinese: '后端阀' | English: 'GVB '
  1049 = 'GVB ALL CL' | Chinese: 'GVB 全关' | English: 'GVB ALL CL'
  1306 = 'GVB ALL OP' | Chinese: 'GVB 全开' | English: 'GVB ALL OP'
  2693 = 'He(500)'
  1792 = 'HI'
  1937 = 'Hide Log Page' | Chinese: '隐藏日志' | English: 'Hide Log Page'
  3195 = 'HL:%.1f' | Chinese: 'HL:%.1f' | English: 'HL:%.1f'
  1050 = 'HO'
  1484 = 'HOME' | Chinese: '原点' | English: 'HOME'
  556 = 'HZ' | Chinese: 'HZ' | English: 'HZ'
  2189 = 'I:%d' | Chinese: 'I:%d' | English: 'I:%d'
  2021 = 'IN' | Chinese: '工作位' | English: 'IN'
  1852 = 'INC' | Chinese: '加' | English: 'INC'
  331 = 'Information' | Chinese: 'Information' | English: 'Information'
  3323 = 'Input' | Chinese: 'Input' | English: 'Input'
  3271 = 'IO' | Chinese: 'IO' | English: 'IO'
  1930 = 'IP & Port'
  2554 = 'ISO. Valve' | Chinese: 'PDV真空阀' | English: 'ISO.Valve'
  2028 = 'ISO.VALVE' | Chinese: 'ISO阀' | English: 'ISO.Gauge'
  361 = 'L:%d'
  860 = 'LIFT PIN' | Chinese: '顶针' | English: 'LIFT PIN'
  1311 = 'LL LID' | Chinese: 'LL盖检测' | English: 'LL LID'
  1222 = 'LL VENT' | Chinese: 'LL破空阀' | English: 'LL VENT'
  529 = 'LOAD' | Chinese: 'LOAD' | English: 'LOAD'
  1413 = 'Load Config' | Chinese: '加载配置' | English: 'Load Config'
  574 = 'LOAD LOCK' | Chinese: '上料锁' | English: 'LOAD LOCK'
  1029 = 'Load Lock Vent' | Chinese: '上料腔破空' | English: 'Load Lock Vent'
  2814 = 'Load Wafer' | Chinese: '上晶圆' | English: 'Load Wafer'
  662 = 'Local IP:' | Chinese: '本地IP:' | English: 'Local IP:'
  2598 = 'Local Port:' | Chinese: '本地端口:' | English: 'Local Port:'
  686 = 'LOG' | Chinese: '日志' | English: 'LOG'
  1786 = 'Machine Vent' | Chinese: '整机破空' | English: 'Machine Pump'
  2276 = 'Manual' | Chinese: '手动' | English: 'Manual'
  812 = 'Max Page' | Chinese: '最大页' | English: 'Max Page'
  1860 = 'MFC'
  2176 = 'MODE' | Chinese: '模式' | English: 'MODE'
  1003 = 'mToor'
  2996 = 'mTorr'
  1322 = 'MV:%d' | Chinese: 'MV:%d' | English: 'MV:%d'
  497 = 'N'
  907 = 'N2(50)'
  965 = 'Next' | Chinese: 'Next' | English: 'Next'
  1221 = 'NON'
  1196 = 'None' | Chinese: 'None' | English: 'None'
  2107 = 'NORMAL' | Chinese: '正常' | English: 'NORMAL'
  1576 = 'NorSw'
  2529 = 'Note View' | Chinese: '操作提示' | English: 'Note View'
  3200 = 'O2(10)'
  166 = 'O2(100)'
  741 = 'OK' | Chinese: '确认' | English: 'OK'
  4365 = 'OpCd'
  619 = 'OpEN'
  525 = 'OPEN' | Chinese: '打开' | English: 'OPEN'
  2129 = 'Open' | Chinese: '打开' | English: 'Open'
  1452 = 'Operator' | Chinese: '操作' | English: 'Operator'
  3393 = 'operator' | Chinese: '操作员' | English: 'operator'
  3519 = 'Other Par' | Chinese: '其他配置' | English: 'Other_Par'
  2844 = 'OT_1'
  2337 = 'OT_2'
  2543 = 'OT_3'
  1107 = 'Output' | Chinese: 'Output' | English: 'Output'
  1249 = 'P'
  1324 = 'P:%d' | Chinese: 'P:%d' | English: 'P:%d'
  828 = 'Page' | Chinese: 'Page' | English: 'Page'
  1505 = 'PARAMETERS OF THEN SELECTED RECIPE' | Chinese: '所选配方参数' | English: 'PARAMETERS OF THE SELECTED RECIPE'
  1298 = 'PASHE'
  588 = 'Pause' | Chinese: '暂停' | English: 'Pause'
  948 = 'PDV' | Chinese: 'PDV' | English: 'PDV'
  483 = 'PDV IP:'
  1477 = 'PDV Port:'
  1001 = 'Please keep pressing to trigger' | Chinese: 'Please keep pressing to trigger' | English: 'Please keep pressing to trigger'
  2040 = 'Please keep pressing to trigger the absolute motion loop' | Chinese: 'Please keep pressing to trigger the absolute motion loop' | English: 'Please keep pressing to trigger the absolute motion loop'
  2858 = 'Please keep pressing to trigger the relative motion loop' | Chinese: 'Please keep pressing to trigger the relative motion loop' | English: 'Please keep pressing to trigger the relative motion loop'
  1916 = 'POS.' | Chinese: '位置' | English: 'POS.'
  870 = 'POSITION' | Chinese: '位置' | English: 'POSITION'
  2474 = 'POU Run Log Show:' | Chinese: '程序运行日志:' | English: 'POU Run Log Show'
  1451 = 'POWER' | Chinese: '启动' | English: 'POWER'
  887 = 'POWER RF' | Chinese: '下电极源' | English: 'POWER RF'
  1442 = 'Power RF' | Chinese: '下电极源' | English: 'Power RF'
  2719 = 'Power RF IP:'
  1947 = 'Power RF Port:'
  239 = 'PowerEN' | Chinese: 'PowerEN' | English: 'PowerEN'
  3178 = 'PRE'
  1820 = 'PRE.' | Chinese: '压力' | English: 'PRE.'
  2715 = 'PRESET'
  171 = 'PRF'
  591 = 'PTPErrID' | Chinese: 'PTPErrID' | English: 'PTPErrID'
  1977 = 'PV' | Chinese: 'PV' | English: 'PV'
  71 = 'PV POS.' | Chinese: '反馈位置' | English: 'PV POS.'
  685 = 'PV PRE.' | Chinese: '压力' | English: 'PV PRE.'
  5189 = 'PV:%.1f'
  161 = 'Recipe' | Chinese: '配方' | English: 'Recipe'
  610 = 'RECIPE NAME' | Chinese: '配方名' | English: 'RECIPE NAME'
  3036 = 'record' | Chinese: '记录' | English: 'record'
  2022 = 'REF. POWER' | Chinese: '反射功率' | English: 'REF. POWER'
  321 = 'REM. TIME' | Chinese: '剩余时间' | English: 'REM. TIME'
  1082 = 'RemainTime:%d s' | Chinese: '剩余时间:%d 秒' | English: 'RemainTime:%d s'
  2425 = 'Reset' | Chinese: '复位' | English: 'Reset'
  1305 = 'RetCd'
  184 = 'RetEN' | Chinese: 'RetEN' | English: 'RetEN'
  180 = 'RetSw' | Chinese: 'RetSw' | English: 'RetSw'
  592 = 'RF Co-Control' | Chinese: 'RF共同控制' | English: 'RF Co-Control'
  655 = 'RF DC BIAS' | Chinese: '偏压' | English: 'RF DC BIAS'
  1110 = 'ROUGH\nVALVE' | Chinese: '粗抽阀' | English: 'ROUGH\nVALVE'
  1676 = 'Rough Pump' | Chinese: '粗抽' | English: 'Rough Pump'
  2733 = 'Runing' | Chinese: '运行' | English: 'Runing'
  1675 = 'S'
  2711 = 'Save Changes' | Chinese: '变更' | English: 'Save Change'
  2690 = 'Save Config' | Chinese: '保存配置' | English: 'Save Config'
  434 = 'Save the current info' | Chinese: 'Save the current info' | English: 'Save the current info'
  2373 = 'Sccm'
  2102 = 'SD:%d'
  2199 = 'SELECT RECIPE' | Chinese: '配方选择' | English: 'SELECT RECIPE'
  1414 = 'SET' | Chinese: '设置' | English: 'SET'
  48 = 'SET POINT' | Chinese: '目标值' | English: 'Set Point'
  450 = 'SET POINT (Max)\n(sccm)' | Chinese: '目标值(最大)\n(sccm)' | English: 'SET POINT(Max)\n(sccm)'
  3128 = 'SET TIME' | Chinese: '时间设置' | English: 'SET TIME'
  3300 = 'Set:%.1f' | Chinese: '设置:%.1f' | English: 'Set:%.1f'
  3117 = 'SF6(200)'
  1526 = 'Show Log Page' | Chinese: '显示日志' | English: 'Show Log Page'
  24 = 'SI:%d' | Chinese: 'SI:%d' | English: 'SI:%d'
  578 = 'SLOW\nVALVE' | Chinese: '预抽阀' | English: 'SLOW\nPUM'
  1064 = 'SMV:%d' | Chinese: 'SMV:%d' | English: 'SMV:%d'
  2050 = 'SOURCE RF' | Chinese: '源RF' | English: 'SOURCE RF'
  1715 = 'Source RF' | Chinese: '源RF' | English: 'Source RF'
  1683 = 'Source RF IP:'
  2025 = 'Source RF Port:'
  678 = 'SP:%d' | Chinese: 'SP:%d' | English: 'SP:%d'
  1817 = 'SPEED' | Chinese: '转速' | English: 'SPEED'
  585 = 'SRF'
  1021 = 'START' | Chinese: '启动' | English: 'START'
  1002 = 'Start' | Chinese: '启动' | English: 'Start'
  179 = 'Status' | Chinese: 'Status' | English: 'Status'
  1784 = 'STATUS' | Chinese: '状态' | English: 'STATUS'
  2455 = 'Stop' | Chinese: '停止' | English: 'Stop'
  1632 = 'STOP' | Chinese: '停止' | English: 'STOP'
  3303 = 'SV:%.1f'
  2460 = 'T1'
  2366 = 'T2'
  4036 = 'T:%.1f℃'
  3004 = 'TEMP' | Chinese: '温度' | English: 'TEMP'
  848 = 'Temp.' | Chinese: '温度' | English: 'Temp.'
  330 = 'Time' | Chinese: 'Time' | English: 'Time'
  2190 = 'TIME' | Chinese: '时间' | English: 'TIME'
  2583 = 'Tips for action'
  1236 = 'Torr'
  5 = 'TURBO PUM' | Chinese: '分子泵' | English: 'TURBO PUM'
  3032 = 'TURBO PUM TAIL' | Chinese: '分子泵尾排' | English: 'TURBO PUM TAIL'
  2380 = 'UnLoad Wafer' | Chinese: '下晶圆' | English: 'UnLoad Wafer'
  1420 = 'User' | Chinese: '用户' | English: 'User'
  134 = 'V' | Chinese: 'V' | English: 'V'
  4141 = 'V:%.1frpm'
  296 = 'V:%d'
  1009 = 'Vent Valve' | Chinese: '破空阀' | English: 'Vent Valve'
  1822 = 'Ver:%s'
  1756 = 'W'
  2169 = 'Wafer In Chamber' | Chinese: '晶圆在腔体内' | English: 'Wafer In Chamber'
  2251 = 'WAFER ON ARM' | Chinese: '晶圆检测' | English: 'WAFER ON ARM'
  2256 = 'Welcome,%s' | Chinese: '欢迎，%s' | English: 'Welcome,%s'
  2299 = '×'
  1475 = '℃' | Chinese: '℃' | English: '℃'
  579 = '√'
  4025 = '伸出/吸' | Chinese: '伸出/吸' | English: 'Extend/Vacuum'
  2437 = '使能' | Chinese: '使能' | English: 'Enable'
  10 = '停止' | Chinese: '停止' | English: 'Stop'
  1686 = '允许正向运动' | Chinese: '允许正向运动' | English: 'Enable Forward'
  6032 = '允许负向运动' | Chinese: '允许负向运动' | English: 'Enable Backward'
  2793 = '分子泵' | Chinese: '分子泵' | English: 'TB'
  2541 = '到位等待时间 [ms]:' | Chinese: '到位等待时间 [ms]:' | English: 'Arrived Wait Time [ms]:'
  3023 = '前级阀' | Chinese: '前级阀' | English: 'ForLineValve'
  750 = '原点' | Chinese: '原点' | English: 'HomeSensor'
  5437 = '原点状态:' | Chinese: '原点状态:' | English: 'Homed Status:'
  2935 = '参数设置说明' | Chinese: '参数设置说明' | English: 'Parameter Setting Explain'
  897 = '启动' | Chinese: '启动' | English: 'Start'
  9987 = '回原' | Chinese: '回原' | English: 'Home'
  3911 = '回原循环' | Chinese: '回原循环' | English: 'Homing Loop'
  2815 = '回原正常速度 [mm/s]:' | Chinese: '回原正常速度 [mm/s]:' | English: 'Home Normal Speed [mm/s]:'
  7285 = '回原爬行速度[mm/s]:' | Chinese: '回原爬行速度[mm/s]:' | English: 'Home Slow Speed [mm/s]:'
  967 = '复位' | Chinese: '复位' | English: 'Reset'
  1228 = '定位速度设置 [mm/s]' | Chinese: '定位速度设置 [mm/s]' | English: 'Vel Speed [mm/s]'
  7878 = '实际位置 [mm]' | Chinese: '实际位置 [mm]' | English: 'Actual Pos [mm]'
  9652 = '实际速度 [mm/s]' | Chinese: '实际速度 [mm/s]' | English: 'Actual Vel [mm/s]'
  7164 = '往返运动速度 [mm/s]:' | Chinese: '往返运动速度 [mm/s]:' | English: 'Loop Velocity [mm/s]:'
  8523 = '循环次数:' | Chinese: '循环次数:' | English: 'Loop Times:'
  2615 = '快抽阀' | Chinese: '快抽阀' | English: 'Fast Valve'
  1823 = '手动加热' | Chinese: '手动加热' | English: 'Manual Het'
  9121 = '暂停' | Chinese: '暂停' | English: 'Pause'
  1589 = '更改密码' | Chinese: '更改密码' | English: 'Change Password'
  1230 = '机械泵' | Chinese: '机械泵' | English: 'Machine Pum'
  1898 = '欢迎，请点击右上角登陆\n界面或登录后选择相应功\n能进行操作' | Chinese: '欢迎，请点击右上角登陆\n界面或登录后选择相应功\n能进行操作' | English: 'Welcome, please click on the login screen\n in the upper right corner \nor \nselect the corresponding function after logging in'
  519 = '正向/反向' | Chinese: '正向/反向' | English: 'Positive/Negative'
  3927 = '正向软限位 [mm]:' | Chinese: '正向软限位 [mm]:' | English: 'Positive Soft Limit [mm]:'
  4624 = '正限位' | Chinese: '正限位' | English: 'Positive Sensor'
  2155 = '水冷机' | Chinese: '水冷机' | English: 'Chiller'
  7519 = '点动' | Chinese: '点动' | English: 'Jog'
  576 = '点动速度设置 [mm/s]' | Chinese: '点动速度设置 [mm/s]' | English: 'Jog Velocity [mm/s]'
  814 = '电极升降台' | Chinese: '电极升降台' | English: 'Electrode'
  1881 = '登        入' | Chinese: '登        入' | English: 'LogIn'
  2170 = '登        出' | Chinese: '登        出' | English: 'LogOut'
  1291 = '相对定位位置设置 [mm]' | Chinese: '相对定位位置设置 [mm]' | English: 'Relative Position [mm]'
  195 = '相对循环' | Chinese: '相对循环' | English: 'RelativeLoop'
  10873 = '相对模式' | Chinese: '相对模式' | English: 'RelativeMode'
  1553 = '禁止' | Chinese: '禁止' | English: 'Abandon'
  693 = '管        理' | Chinese: '管        理' | English: 'Config'
  1141 = '粗抽阀' | Chinese: '粗抽阀' | English: 'Rough Valve'
  8848 = '终点位置[mm]:' | Chinese: '终点位置[mm]:' | English: 'End Position[mm]:'
  5283 = '绝对定位位置设置 [mm]' | Chinese: '绝对定位位置设置 [mm]' | English: 'Absolute Position [mm]'
  3673 = '绝对循环' | Chinese: '绝对循环' | English: 'Absolute Loop'
  3724 = '绝对模式' | Chinese: '绝对模式' | English: 'AbsoluteMode'
  7449 = '缩回/吹' | Chinese: '缩回/吹' | English: 'Retract/Break'
  632 = '自动加热' | Chinese: '自动加热' | English: 'Auto Heat'
  189 = '自学习' | Chinese: '自学习' | English: 'Auto Learn'
  6295 = '设零' | Chinese: '设零' | English: 'Set to Zero'
  2786 = '负向软限位 [mm]:' | Chinese: '负向软限位 [mm]:' | English: 'Negative Soft Limit [mm]:'
  4462 = '负限位' | Chinese: '负限位' | English: 'Negetive Sensor'
  5037 = '起点位置 [mm]:' | Chinese: '起点位置 [mm]:' | English: 'Start Position [mm]:'
  3352 = '输入' | Chinese: '输入' | English: 'Input'
  3910 = '输出' | Chinese: '输出' | English: 'Output'
  6480 = '速度模式' | Chinese: '速度模式' | English: 'VelocityMode'
  2953 = '钟摆阀' | Chinese: '钟摆阀' | English: 'PDV'
  3427 = '需切换界面左上角控制模式为“配置模式”，根据参数栏\n\n左上方提示内容及其设置框说明标题，设置相应的参数并按\n\n“保存配置”按钮3秒以上，直到右侧黄灯闪烁\n\n设置完成参数后需根据相应需求选择对应控制模式' | Chinese: '需切换界面左上角控制模式为“配置模式”，根据参数栏\n\n左上方提示内容及其设置框说明标题，设置相应的参数并按\n\n“保存配置”按钮3秒以上，直到右侧黄灯闪烁\n\n设置完成参数后需根据相应需求选择对应控制模式' | English: "Switch control mode to Configuration Mode.\nPress the 'Save' button for more than 3 seconds until the yellow light on the right flashes"
  406 = '顶针' | Chinese: '顶针' | English: 'LiftPin'
  1344 = '预抽阀' | Chinese: '预抽阀' | English: 'Rough Valve'
END_TEXTLIST

// ---- POUs/BaseModule/ActionModule/cylinderModule/visu/cylinderModuleVisu.TcVIS
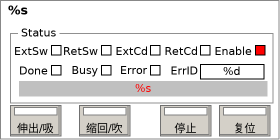
VISUALIZATION cylinderModuleVisu  // 280x140
VAR_IN_OUT
	userData: CylinderModuleHMI;
END_VAR
    Button (10,105 51x31), "伸出/吸", input disabled if: NOT userData.HMIEnable
        tap userData.extend
    Rectangle (14,107 43x8), colour toggle: userData.extRelay
    GroupBox (10,25 263x78), "Status"
        Label (54,20 37x13), "RetSw"
        Label (4,20 37x13), "ExtSw"
        RoundedRectangle (41,20 10x10), colour toggle: userData.extAprSw
        RoundedRectangle (91,20 10x10), colour toggle: userData.retAprSw
        RoundedRectangle (41,40 10x10), colour toggle: userData.done
        RoundedRectangle (245,20 10x10), colour toggle: userData.enable
        RoundedRectangle (91,40 10x10), colour toggle: userData.busy
        RoundedRectangle (140,40 10x10), colour toggle: userData.error
        Rectangle (190,39 64x15), "%d", text variable: userData.errID
        Label (104,20 37x13), "ExtCd"
        RoundedRectangle (140,20 10x10), colour toggle: userData.extcondition
        Label (154,20 37x13), "RetCd"
        RoundedRectangle (190,20 10x10), colour toggle: userData.retcondition
        Rectangle (9,56 248x15), "%s", text variable: userData.errTXT
        Label (206,20 39x13), "Enable"
        Label (158,39 33x14), "ErrID"
        Label (110,39 30x13), "Error"
        Label (61,39 30x13), "Busy"
        Label (8,38 33x16), "Done"
    Button (79,105 51x31), "缩回/吹", input disabled if: NOT userData.HMIEnable
        tap userData.retract
    Rectangle (83,107 43x8), colour toggle: userData.retRelay
    Button (219,105 51x31), "复位"
        tap userData.reset
    Rectangle (223,107 43x8), colour toggle: userData.error
    Rectangle (5,0 267x20), "%s", text variable: userData.nameTXT
    Button (160,105 51x31), "停止"
        tap userData.stop
    Rectangle (164,107 43x8)
END_VISUALIZATION

// ---- POUs/BaseModule/ActionModule/cylinderModule/visu/cylinderModuleVisu_1.TcVIS
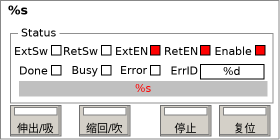
VISUALIZATION cylinderModuleVisu_1  // 280x140
VAR_IN_OUT
	userData: CylinderModuleHMI;
END_VAR
    Button (10,105 51x31), "伸出/吸", input disabled if: NOT userData.HMIEnable
        tap userData.extend
    Rectangle (14,107 43x8), colour toggle: userData.extRelay
    GroupBox (10,25 263x78), "Status"
        Label (54,20 37x13), "RetSw"
        Label (4,20 37x13), "ExtSw"
        RoundedRectangle (41,20 10x10), colour toggle: userData.extAprSw
        RoundedRectangle (91,20 10x10), colour toggle: userData.retAprSw
        RoundedRectangle (41,40 10x10), colour toggle: userData.done
        RoundedRectangle (245,20 10x10), colour toggle: userData.enable
        RoundedRectangle (91,40 10x10), colour toggle: userData.busy
        RoundedRectangle (140,40 10x10), colour toggle: userData.error
        Rectangle (190,39 64x15), "%d", text variable: userData.errID
        Label (104,20 37x13), "ExtEN"
        RoundedRectangle (140,20 10x10), colour toggle: userData.enableExt
        Label (154,20 37x13), "RetEN"
        RoundedRectangle (190,20 10x10), colour toggle: userData.enableRet
        Rectangle (9,56 248x15), "%s", text variable: userData.errTXT
        Label (206,20 39x13), "Enable"
        Label (158,39 33x14), "ErrID"
        Label (110,39 30x13), "Error"
        Label (61,39 30x13), "Busy"
        Label (8,38 33x16), "Done"
    Button (79,105 51x31), "缩回/吹", input disabled if: NOT userData.HMIEnable
        tap userData.retract
    Rectangle (83,107 43x8), colour toggle: userData.retRelay
    Button (219,105 51x31), "复位"
        tap userData.reset
    Rectangle (223,107 43x8), colour toggle: userData.error
    Rectangle (5,0 267x20), "%s", text variable: userData.nameTXT
    Button (160,105 51x31), "停止"
        tap userData.stop
    Rectangle (164,107 43x8)
END_VISUALIZATION

// ---- POUs/BaseModule/ActionModule/HEATModule/visu/HeatModuleVisu.TcVIS
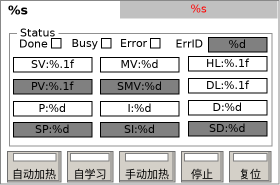
VISUALIZATION HeatModuleVisu  // 280x185
VAR_IN_OUT
	userData:HEATModuleHMI;
END_VAR
    Button (7,151 54x31), "自动加热", input disabled if: NOT userData.HMIEnable
        tap userData.heat
    Rectangle (13,153 43x8), colour toggle: userData.busy
    GroupBox (9,25 263x121), "Status"
        RoundedRectangle (42,13 10x10), colour toggle: userData.done
        RoundedRectangle (92,13 10x10), colour toggle: userData.busy
        RoundedRectangle (141,13 10x10), colour toggle: userData.error
        Rectangle (199,12 59x15), "%d", text variable: userData.errID, input disabled if: true
        Label (164,12 33x14), "ErrID"
        Label (111,12 30x13), "Error"
        Label (62,12 30x13), "Busy"
        Label (9,11 33x16), "Done"
        Rectangle (4,32 79x15), "SV:%.1f", text variable: userData.para_SV
            OnMouseClick: write the text variable via Default, min -10, max 300
        Rectangle (4,54 79x15), "PV:%.1f", text variable: userData.status_PV, input disabled if: true
        Rectangle (91,54 79x15), "SMV:%d", text variable: userData.status_MV, input disabled if: true
        Rectangle (179,53 79x15), "DL:%.1f", text variable: userData.para_LLimit
            OnMouseClick: write the text variable via Default, min -10, max 300
        Rectangle (4,76 79x15), "P:%d", text variable: userData.para_P
            OnMouseClick: write the text variable via Default, min -10, max 300
        Rectangle (91,76 79x15), "I:%d", text variable: userData.para_I
            OnMouseClick: write the text variable via Default, min -10, max 300
        Rectangle (4,97 79x15), "SP:%d", text variable: userData.status_P, input disabled if: true
    Button (67,151 46x31), "自学习", input disabled if: NOT userData.HMIEnable
        tap userData.ATLearning
    Rectangle (70,153 39x8)
    Button (229,151 42x31), "复位"
        tap userData.reset
    Rectangle (233,153 34x8), colour toggle: userData.error
    Rectangle (5,0 112x20), "%s", text variable: userData.nameTXT
    Button (119,151 56x31), "手动加热", input disabled if: false
        tap userData.manuleHeat
    Rectangle (125,153 43x8)
    Button (181,151 42x31), "停止"
        tap userData.stop
    Rectangle (184,153 34x8), colour toggle: userData.stop
    Rectangle (120,0 157x18), "%s", text variable: userData.errTXT
    Rectangle (100,57 79x15), "MV:%d", text variable: userData.para_Manual_MV
        OnMouseClick: write the text variable via Default, min -10, max 300
    Rectangle (188,56 79x15), "HL:%.1f", text variable: userData.para_HLimit
        OnMouseClick: write the text variable via Default, min -10, max 300
    Rectangle (188,100 79x15), "D:%d", text variable: userData.para_D
        OnMouseClick: write the text variable via Default, min -10, max 300
    Rectangle (100,122 79x15), "SI:%d", text variable: userData.status_I, input disabled if: true
    Rectangle (188,121 79x15), "SD:%d", text variable: userData.status_D, input disabled if: true
END_VISUALIZATION

